LIN {X 0,Y 348.541,Z 887.712,A -85,B 0,C 180,E1 25758,E2 25758} C_VEL
LIN {X 0,Y 309.674,Z 947.389,A -85,B 0,C 180,E1 25764.214,E2 25764.214} C_VEL
LIN {X 0,Y 266.676,Z 997.893,A -85,B 0,C 180,E1 25773.835,E2 25773.835} C_VEL
LIN {X 0,Y 228.973,Z 1035.675,A -85,B 0,C 180,E1 25788.528,E2 25788.528} C_VEL
LIN {X 0,Y 208.44,Z 1057.583,A -85,B 0,C 180,E1 25806.415,E2 25806.415} C_VEL
LIN {X 0,Y 203.021,Z 1066.413,A -85,B 0,C 180,E1 25823.568,E2 25823.568} C_VEL
LIN {X 0,Y 203.129,Z 1067.072,A -85,B 0,C 180,E1 25836.43,E2 25836.43} C_VEL
LIN {X 0,Y 210.406,Z 1057.864,A -85,B 0,C 180,E1 25856.198,E2 25856.198} C_VEL
LIN {X 0,Y 222.858,Z 1046.1,A -85,B 0,C 180,E1 25867.529,E2 25867.529} C_VEL
LIN {X 0,Y 229.777,Z 1035.055,A -85,B 0,C 180,E1 25875.914,E2 25875.914} C_VEL
LIN {X 0,Y 272.123,Z 997.636,A -85,B 0,C 180,E1 25889.741,E2 25889.741} C_VEL
LIN {X 0,Y 318.781,Z 947.378,A -85,B 0,C 180,E1 25898.568,E2 25898.568} C_VEL
LIN {X 0,Y 352.077,Z 901.57,A -85,B 0,C 180,E1 25903.055,E2 25903.055} C_VEL
LIN {X 0,Y 353.093,Z 885.679,A -85,B 0,C 180,E1 25911.32,E2 25911.32} C_VEL
LIN {X 0,Y 353.625,Z 880.392,A -85,B 0,C 180,E1 25918.744,E2 25918.744} C_VEL
LIN {X 0,Y 352.671,Z 887.548,A -85,B 0,C 180,E1 25927.391,E2 25927.391} C_VEL
LIN {X 0,Y 350.818,Z 902.517,A -85,B 0,C 180,E1 25934.441,E2 25934.441} C_VEL
LIN {X 0,Y 306.477,Z 960.307,A -85,B 0,C 180,E1 25940.703,E2 25940.703} C_VEL
LIN {X 0,Y 260.092,Z 1006.735,A -85,B 0,C 180,E1 25950.78,E2 25950.78} C_VEL
LIN {X 0,Y 220.914,Z 1039.817,A -85,B 0,C 180,E1 25966.109,E2 25966.109} C_VEL
LIN {X 0,Y 199.649,Z 1057.963,A -85,B 0,C 180,E1 25985.307,E2 25985.307} C_VEL
LIN {X 0,Y 194.828,Z 1063.462,A -85,B 0,C 180,E1 26003.294,E2 26003.294} C_VEL
LIN {X 0,Y 195.704,Z 1061.786,A -85,B 0,C 180,E1 26016.673,E2 26016.673} C_VEL
LIN {X 0,Y 206.346,Z 1048.693,A -85,B 0,C 180,E1 26037.341,E2 26037.341} C_VEL
LIN {X 0,Y 236.758,Z 1019.964,A -85,B 0,C 180,E1 26055.856,E2 26055.856} C_VEL
LIN {X 0,Y 278.852,Z 977.829,A -85,B 0,C 180,E1 26068.386,E2 26068.386} C_VEL
LIN {X 0,Y 322.725,Z 923.382,A -85,B 0,C 180,E1 26076.469,E2 26076.469} C_VEL
LIN {X 0,Y 342.393,Z 892.633,A -85,B 0,C 180,E1 26079.429,E2 26079.429} C_VEL
LIN {X 0,Y 343.314,Z 872.383,A -85,B 0,C 180,E1 26087.906,E2 26087.906} C_VEL
LIN {X 0,Y 343.606,Z 863.388,A -85,B 0,C 180,E1 26096.228,E2 26096.228} C_VEL
LIN {X 0,Y 343.762,Z 863.668,A -85,B 0,C 180,E1 26101.292,E2 26101.292} C_VEL
LIN {X 0,Y 343.852,Z 876.291,A -85,B 0,C 180,E1 26110.841,E2 26110.841} C_VEL
LIN {X 0,Y 342.839,Z 893.969,A -85,B 0,C 180,E1 26117.448,E2 26117.448} C_VEL
LIN {X 0,Y 301.371,Z 953.407,A -85,B 0,C 180,E1 26123.657,E2 26123.657} C_VEL
LIN {X 0,Y 257.23,Z 1002.52,A -85,B 0,C 180,E1 26133.7,E2 26133.7} C_VEL
LIN {X 0,Y 219.56,Z 1038.628,A -85,B 0,C 180,E1 26148.996,E2 26148.996} C_VEL
LIN {X 0,Y 199.54,Z 1059.052,A -85,B 0,C 180,E1 26167.669,E2 26167.669} C_VEL
LIN {X 0,Y 195.018,Z 1066.321,A -85,B 0,C 180,E1 26183.303,E2 26183.303} C_VEL
LIN {X 0,Y 195.122,Z 1066.998,A -85,B 0,C 180,E1 26196.695,E2 26196.695} C_VEL
LIN {X 0,Y 202.007,Z 1058.771,A -85,B 0,C 180,E1 26215.932,E2 26215.932} C_VEL
LIN {X 0,Y 229.777,Z 1035.055,A -85,B 0,C 180,E1 26235.914,E2 26235.914} C_VEL
LIN {X 0,Y 239.937,Z 1022.061,A -85,B 0,C 180,E1 26243.59,E2 26243.59} C_VEL
LIN {X 0,Y 287.569,Z 978.627,A -85,B 0,C 180,E1 26255.332,E2 26255.332} C_VEL
LIN {X 0,Y 334.687,Z 923.76,A -85,B 0,C 180,E1 26262.455,E2 26262.455} C_VEL
LIN {X 0,Y 347.143,Z 905.9,A -85,B 0,C 180,E1 26263.988,E2 26263.988} C_VEL
LIN {X 0,Y 348.572,Z 891.02,A -85,B 0,C 180,E1 26272.467,E2 26272.467} C_VEL
LIN {X 0,Y 349.117,Z 887.018,A -85,B 0,C 180,E1 26278.727,E2 26278.727} C_VEL
LIN {X 0,Y 347.911,Z 894.709,A -85,B 0,C 180,E1 26287.711,E2 26287.711} C_VEL
LIN {X 0,Y 345.687,Z 907.135,A -85,B 0,C 180,E1 26293.499,E2 26293.499} C_VEL
LIN {X 0,Y 300.619,Z 963.408,A -85,B 0,C 180,E1 26299.715,E2 26299.715} C_VEL
LIN {X 0,Y 253.465,Z 1008.739,A -85,B 0,C 180,E1 26309.829,E2 26309.829} C_VEL
LIN {X 0,Y 212.875,Z 1041.423,A -85,B 0,C 180,E1 26325.724,E2 26325.724} C_VEL
LIN {X 0,Y 191.326,Z 1058.749,A -85,B 0,C 180,E1 26345.704,E2 26345.704} C_VEL
LIN {X 0,Y 186.807,Z 1063.535,A -85,B 0,C 180,E1 26363.005,E2 26363.005} C_VEL
LIN {X 0,Y 187.75,Z 1061.89,A -85,B 0,C 180,E1 26376.957,E2 26376.957} C_VEL
LIN {X 0,Y 197.993,Z 1049.851,A -85,B 0,C 180,E1 26397.274,E2 26397.274} C_VEL
LIN {X 0,Y 227.623,Z 1023.387,A -85,B 0,C 180,E1 26415.862,E2 26415.862} C_VEL
LIN {X 0,Y 270.255,Z 982.815,A -85,B 0,C 180,E1 26428.834,E2 26428.834} C_VEL
LIN {X 0,Y 315.398,Z 929.408,A -85,B 0,C 180,E1 26437.172,E2 26437.172} C_VEL
LIN {X 0,Y 337.365,Z 896.845,A -85,B 0,C 180,E1 26440.31,E2 26440.31} C_VEL
LIN {X 0,Y 338.999,Z 877.413,A -85,B 0,C 180,E1 26449.059,E2 26449.059} C_VEL
LIN {X 0,Y 340.014,Z 868.942,A -85,B 0,C 180,E1 26458.749,E2 26458.749} C_VEL
LIN {X 0,Y 339.391,Z 878.655,A -85,B 0,C 180,E1 26468.385,E2 26468.385} C_VEL
LIN {X 0,Y 338.245,Z 897.158,A -85,B 0,C 180,E1 26476.407,E2 26476.407} C_VEL
LIN {X 0,Y 294.973,Z 956.872,A -85,B 0,C 180,E1 26482.735,E2 26482.735} C_VEL
LIN {X 0,Y 249.571,Z 1005.349,A -85,B 0,C 180,E1 26493.014,E2 26493.014} C_VEL
LIN {X 0,Y 211.634,Z 1040.081,A -85,B 0,C 180,E1 26508.542,E2 26508.542} C_VEL
LIN {X 0,Y 190.684,Z 1060.513,A -85,B 0,C 180,E1 26529.032,E2 26529.032} C_VEL
LIN {X 0,Y 186.999,Z 1067.028,A -85,B 0,C 180,E1 26547.677,E2 26547.677} C_VEL
LIN {X 0,Y 187.65,Z 1065.942,A -85,B 0,C 180,E1 26561.657,E2 26561.657} C_VEL
LIN {X 0,Y 200.399,Z 1053.731,A -85,B 0,C 180,E1 26583.213,E2 26583.213} C_VEL
LIN {X 0,Y 234.442,Z 1026.63,A -85,B 0,C 180,E1 26601.681,E2 26601.681} C_VEL
LIN {X 0,Y 239.937,Z 1022.061,A -85,B 0,C 180,E1 26603.59,E2 26603.59} C_VEL
LIN {X 0,Y 253.584,Z 1007.011,A -85,B 0,C 180,E1 26610.365,E2 26610.365} C_VEL
LIN {X 0,Y 302.812,Z 959.33,A -85,B 0,C 180,E1 26619.879,E2 26619.879} C_VEL
LIN {X 0,Y 342.323,Z 909.562,A -85,B 0,C 180,E1 26625.257,E2 26625.257} C_VEL
LIN {X 0,Y 344.01,Z 896.36,A -85,B 0,C 180,E1 26633.64,E2 26633.64} C_VEL
LIN {X 0,Y 344.292,Z 894.425,A -85,B 0,C 180,E1 26641.236,E2 26641.236} C_VEL
LIN {X 0,Y 342.35,Z 905.549,A -85,B 0,C 180,E1 26650.211,E2 26650.211} C_VEL
LIN {X 0,Y 340.57,Z 911.466,A -85,B 0,C 180,E1 26652.525,E2 26652.525} C_VEL
LIN {X 0,Y 294.571,Z 966.733,A -85,B 0,C 180,E1 26658.74,E2 26658.74} C_VEL
LIN {X 0,Y 245.604,Z 1011.828,A -85,B 0,C 180,E1 26669.183,E2 26669.183} C_VEL
LIN {X 0,Y 204.818,Z 1043.029,A -85,B 0,C 180,E1 26685.302,E2 26685.302} C_VEL
LIN {X 0,Y 182.092,Z 1060.341,A -85,B 0,C 180,E1 26707.99,E2 26707.99} C_VEL
LIN {X 0,Y 179.012,Z 1063.546,A -85,B 0,C 180,E1 26727.983,E2 26727.983} C_VEL
LIN {X 0,Y 182.801,Z 1057.745,A -85,B 0,C 180,E1 26747.458,E2 26747.458} C_VEL
LIN {X 0,Y 204.643,Z 1038.037,A -85,B 0,C 180,E1 26769.038,E2 26769.038} C_VEL
LIN {X 0,Y 244.88,Z 1003.338,A -85,B 0,C 180,E1 26785.134,E2 26785.134} C_VEL
LIN {X 0,Y 291.96,Z 954.998,A -85,B 0,C 180,E1 26795.357,E2 26795.357} C_VEL
LIN {X 0,Y 332.46,Z 900.578,A -85,B 0,C 180,E1 26801.407,E2 26801.407} C_VEL
LIN {X 0,Y 334.388,Z 883.799,A -85,B 0,C 180,E1 26809.302,E2 26809.302} C_VEL
LIN {X 0,Y 335.804,Z 875.772,A -85,B 0,C 180,E1 26818.733,E2 26818.733} C_VEL
LIN {X 0,Y 334.7,Z 885.63,A -85,B 0,C 180,E1 26828.504,E2 26828.504} C_VEL
LIN {X 0,Y 332.665,Z 901.995,A -85,B 0,C 180,E1 26835.463,E2 26835.463} C_VEL
LIN {X 0,Y 288.685,Z 960.322,A -85,B 0,C 180,E1 26841.778,E2 26841.778} C_VEL
LIN {X 0,Y 242.089,Z 1008.031,A -85,B 0,C 180,E1 26852.263,E2 26852.263} C_VEL
LIN {X 0,Y 202.346,Z 1042.515,A -85,B 0,C 180,E1 26868.897,E2 26868.897} C_VEL
LIN {X 0,Y 181.929,Z 1061.643,A -85,B 0,C 180,E1 26890.525,E2 26890.525} C_VEL
LIN {X 0,Y 178.981,Z 1066.945,A -85,B 0,C 180,E1 26907.573,E2 26907.573} C_VEL
LIN {X 0,Y 180.118,Z 1065.434,A -85,B 0,C 180,E1 26924.076,E2 26924.076} C_VEL
LIN {X 0,Y 196.209,Z 1051.677,A -85,B 0,C 180,E1 26946.797,E2 26946.797} C_VEL
LIN {X 0,Y 233.865,Z 1023.081,A -85,B 0,C 180,E1 26964.828,E2 26964.828} C_VEL
LIN {X 0,Y 253.584,Z 1007.011,A -85,B 0,C 180,E1 26970.365,E2 26970.365} C_VEL
LIN {X 0,Y 269.364,Z 989.826,A -85,B 0,C 180,E1 26976.24,E2 26976.24} C_VEL
LIN {X 0,Y 318.309,Z 938.81,A -85,B 0,C 180,E1 26983.774,E2 26983.774} C_VEL
LIN {X 0,Y 337.204,Z 914.36,A -85,B 0,C 180,E1 26986.015,E2 26986.015} C_VEL
LIN {X 0,Y 339.308,Z 901.839,A -85,B 0,C 180,E1 26994.839,E2 26994.839} C_VEL
LIN {X 0,Y 339.456,Z 900.885,A -85,B 0,C 180,E1 27001.253,E2 27001.253} C_VEL
LIN {X 0,Y 337.059,Z 912.229,A -85,B 0,C 180,E1 27010.344,E2 27010.344} C_VEL
LIN {X 0,Y 334.418,Z 917.307,A -85,B 0,C 180,E1 27011.64,E2 27011.64} C_VEL
LIN {X 0,Y 286.994,Z 971.724,A -85,B 0,C 180,E1 27017.993,E2 27017.993} C_VEL
LIN {X 0,Y 237.199,Z 1015.272,A -85,B 0,C 180,E1 27028.634,E2 27028.634} C_VEL
LIN {X 0,Y 195.356,Z 1045.415,A -85,B 0,C 180,E1 27045.683,E2 27045.683} C_VEL
LIN {X 0,Y 174.467,Z 1060.395,A -85,B 0,C 180,E1 27066.974,E2 27066.974} C_VEL
LIN {X 0,Y 170.98,Z 1063.623,A -85,B 0,C 180,E1 27087.959,E2 27087.959} C_VEL
LIN {X 0,Y 174.832,Z 1058.138,A -85,B 0,C 180,E1 27107.671,E2 27107.671} C_VEL
LIN {X 0,Y 197.219,Z 1039.049,A -85,B 0,C 180,E1 27129.877,E2 27129.877} C_VEL
LIN {X 0,Y 239.003,Z 1004.751,A -85,B 0,C 180,E1 27146.381,E2 27146.381} C_VEL
LIN {X 0,Y 287.218,Z 956.934,A -85,B 0,C 180,E1 27156.585,E2 27156.585} C_VEL
LIN {X 0,Y 327.618,Z 904.456,A -85,B 0,C 180,E1 27162.505,E2 27162.505} C_VEL
LIN {X 0,Y 330.043,Z 888.073,A -85,B 0,C 180,E1 27171.051,E2 27171.051} C_VEL
LIN {X 0,Y 331.379,Z 882.482,A -85,B 0,C 180,E1 27178.716,E2 27178.716} C_VEL
LIN {X 0,Y 330.064,Z 891.717,A -85,B 0,C 180,E1 27188.091,E2 27188.091} C_VEL
LIN {X 0,Y 327.626,Z 906.151,A -85,B 0,C 180,E1 27194.438,E2 27194.438} C_VEL
LIN {X 0,Y 281.995,Z 964.279,A -85,B 0,C 180,E1 27200.882,E2 27200.882} C_VEL
LIN {X 0,Y 234.984,Z 1010.175,A -85,B 0,C 180,E1 27211.35,E2 27211.35} C_VEL
LIN {X 0,Y 194.31,Z 1043.843,A -85,B 0,C 180,E1 27228.446,E2 27228.446} C_VEL
LIN {X 0,Y 174.265,Z 1061.532,A -85,B 0,C 180,E1 27249.632,E2 27249.632} C_VEL
LIN {X 0,Y 170.962,Z 1066.863,A -85,B 0,C 180,E1 27267.459,E2 27267.459} C_VEL
LIN {X 0,Y 171.821,Z 1065.811,A -85,B 0,C 180,E1 27282.748,E2 27282.748} C_VEL
LIN {X 0,Y 186.156,Z 1054.082,A -85,B 0,C 180,E1 27305.526,E2 27305.526} C_VEL
LIN {X 0,Y 223.67,Z 1027.273,A -85,B 0,C 180,E1 27324.723,E2 27324.723} C_VEL
LIN {X 0,Y 269.364,Z 989.826,A -85,B 0,C 180,E1 27336.24,E2 27336.24} C_VEL
LIN {X 0,Y 286.604,Z 970.708,A -85,B 0,C 180,E1 27341.286,E2 27341.286} C_VEL
LIN {X 0,Y 332.201,Z 918.868,A -85,B 0,C 180,E1 27346.947,E2 27346.947} C_VEL
LIN {X 0,Y 334.735,Z 907.351,A -85,B 0,C 180,E1 27356.072,E2 27356.072} C_VEL
LIN {X 0,Y 334.247,Z 908.345,A -85,B 0,C 180,E1 27362.574,E2 27362.574} C_VEL
LIN {X 0,Y 331.472,Z 918.963,A -85,B 0,C 180,E1 27370.395,E2 27370.395} C_VEL
LIN {X 0,Y 282.917,Z 973.223,A -85,B 0,C 180,E1 27376.645,E2 27376.645} C_VEL
LIN {X 0,Y 233.296,Z 1015.235,A -85,B 0,C 180,E1 27386.826,E2 27386.826} C_VEL
LIN {X 0,Y 189.349,Z 1045.482,A -85,B 0,C 180,E1 27403.961,E2 27403.961} C_VEL
LIN {X 0,Y 166.924,Z 1060.449,A -85,B 0,C 180,E1 27425.869,E2 27425.869} C_VEL
LIN {X 0,Y 162.944,Z 1063.699,A -85,B 0,C 180,E1 27447.938,E2 27447.938} C_VEL
LIN {X 0,Y 167.135,Z 1058.253,A -85,B 0,C 180,E1 27468.514,E2 27468.514} C_VEL
LIN {X 0,Y 190.412,Z 1039.655,A -85,B 0,C 180,E1 27491.096,E2 27491.096} C_VEL
LIN {X 0,Y 233.243,Z 1006.068,A -85,B 0,C 180,E1 27507.69,E2 27507.69} C_VEL
LIN {X 0,Y 282.722,Z 958.748,A -85,B 0,C 180,E1 27517.871,E2 27517.871} C_VEL
LIN {X 0,Y 322.812,Z 908.34,A -85,B 0,C 180,E1 27523.646,E2 27523.646} C_VEL
LIN {X 0,Y 325.542,Z 893.675,A -85,B 0,C 180,E1 27531.988,E2 27531.988} C_VEL
LIN {X 0,Y 326.852,Z 889.135,A -85,B 0,C 180,E1 27538.698,E2 27538.698} C_VEL
LIN {X 0,Y 325.154,Z 898.537,A -85,B 0,C 180,E1 27548.214,E2 27548.214} C_VEL
LIN {X 0,Y 322.892,Z 909.93,A -85,B 0,C 180,E1 27553.363,E2 27553.363} C_VEL
LIN {X 0,Y 276.004,Z 967.263,A -85,B 0,C 180,E1 27559.803,E2 27559.803} C_VEL
LIN {X 0,Y 226.78,Z 1013.301,A -85,B 0,C 180,E1 27570.722,E2 27570.722} C_VEL
LIN {X 0,Y 186.449,Z 1045.048,A -85,B 0,C 180,E1 27587.859,E2 27587.859} C_VEL
LIN {X 0,Y 165.492,Z 1062.651,A -85,B 0,C 180,E1 27611.296,E2 27611.296} C_VEL
LIN {X 0,Y 163.159,Z 1067.062,A -85,B 0,C 180,E1 27632.665,E2 27632.665} C_VEL
LIN {X 0,Y 167.989,Z 1062.223,A -85,B 0,C 180,E1 27653.968,E2 27653.968} C_VEL
LIN {X 0,Y 196.071,Z 1043.127,A -85,B 0,C 180,E1 27677.286,E2 27677.286} C_VEL
LIN {X 0,Y 242.567,Z 1009.611,A -85,B 0,C 180,E1 27692.981,E2 27692.981} C_VEL
LIN {X 0,Y 286.604,Z 970.708,A -85,B 0,C 180,E1 27701.286,E2 27701.286} C_VEL
LIN {X 0,Y 304.813,Z 949.598,A -85,B 0,C 180,E1 27705.556,E2 27705.556} C_VEL
LIN {X 0,Y 327.39,Z 922.805,A -85,B 0,C 180,E1 27708.249,E2 27708.249} C_VEL
LIN {X 0,Y 329.635,Z 913.664,A -85,B 0,C 180,E1 27716.011,E2 27716.011} C_VEL
LIN {X 0,Y 329.018,Z 914.821,A -85,B 0,C 180,E1 27722.845,E2 27722.845} C_VEL
LIN {X 0,Y 326.672,Z 923.17,A -85,B 0,C 180,E1 27729.33,E2 27729.33} C_VEL
LIN {X 0,Y 275.725,Z 977.559,A -85,B 0,C 180,E1 27735.748,E2 27735.748} C_VEL
LIN {X 0,Y 223.661,Z 1019.345,A -85,B 0,C 180,E1 27746.502,E2 27746.502} C_VEL
LIN {X 0,Y 179.921,Z 1047.733,A -85,B 0,C 180,E1 27764.241,E2 27764.241} C_VEL
LIN {X 0,Y 159.422,Z 1060.503,A -85,B 0,C 180,E1 27784.655,E2 27784.655} C_VEL
LIN {X 0,Y 154.915,Z 1063.776,A -85,B 0,C 180,E1 27807.919,E2 27807.919} C_VEL
LIN {X 0,Y 159.467,Z 1058.368,A -85,B 0,C 180,E1 27829.439,E2 27829.439} C_VEL
LIN {X 0,Y 186.264,Z 1038.517,A -85,B 0,C 180,E1 27853.787,E2 27853.787} C_VEL
LIN {X 0,Y 231.752,Z 1004.007,A -85,B 0,C 180,E1 27870.108,E2 27870.108} C_VEL
LIN {X 0,Y 282.667,Z 955.853,A -85,B 0,C 180,E1 27879.852,E2 27879.852} C_VEL
LIN {X 0,Y 317.979,Z 912.169,A -85,B 0,C 180,E1 27884.811,E2 27884.811} C_VEL
LIN {X 0,Y 320.895,Z 898.962,A -85,B 0,C 180,E1 27893.239,E2 27893.239} C_VEL
LIN {X 0,Y 322.215,Z 895.711,A -85,B 0,C 180,E1 27898.68,E2 27898.68} C_VEL
LIN {X 0,Y 320.143,Z 905.118,A -85,B 0,C 180,E1 27908.207,E2 27908.207} C_VEL
LIN {X 0,Y 318.121,Z 913.642,A -85,B 0,C 180,E1 27912.264,E2 27912.264} C_VEL
LIN {X 0,Y 269.714,Z 970.668,A -85,B 0,C 180,E1 27918.751,E2 27918.751} C_VEL
LIN {X 0,Y 220.53,Z 1014.822,A -85,B 0,C 180,E1 27929.474,E2 27929.474} C_VEL
LIN {X 0,Y 178.285,Z 1046.464,A -85,B 0,C 180,E1 27947.407,E2 27947.407} C_VEL
LIN {X 0,Y 157.783,Z 1062.539,A -85,B 0,C 180,E1 27970.345,E2 27970.345} C_VEL
LIN {X 0,Y 155.149,Z 1066.988,A -85,B 0,C 180,E1 27992.802,E2 27992.802} C_VEL
LIN {X 0,Y 161.499,Z 1061.503,A -85,B 0,C 180,E1 28016.64,E2 28016.64} C_VEL
LIN {X 0,Y 193.898,Z 1041.055,A -85,B 0,C 180,E1 28040.633,E2 28040.633} C_VEL
LIN {X 0,Y 241.83,Z 1007.483,A -85,B 0,C 180,E1 28055.402,E2 28055.402} C_VEL
LIN {X 0,Y 293.56,Z 961.468,A -85,B 0,C 180,E1 28064.14,E2 28064.14} C_VEL
LIN {X 0,Y 304.813,Z 949.598,A -85,B 0,C 180,E1 28065.556,E2 28065.556} C_VEL
LIN {X 0,Y 315.848,Z 935.192,A -85,B 0,C 180,E1 28068.457,E2 28068.457} C_VEL
LIN {X 0,Y 322.477,Z 926.683,A -85,B 0,C 180,E1 28069.633,E2 28069.633} C_VEL
LIN {X 0,Y 324.901,Z 918.901,A -85,B 0,C 180,E1 28078.633,E2 28078.633} C_VEL
LIN {X 0,Y 322.004,Z 926.631,A -85,B 0,C 180,E1 28087.756,E2 28087.756} C_VEL
LIN {X 0,Y 308.073,Z 943.178,A -85,B 0,C 180,E1 28089.688,E2 28089.688} C_VEL
LIN {X 0,Y 255.938,Z 992.544,A -85,B 0,C 180,E1 28096.864,E2 28096.864} C_VEL
LIN {X 0,Y 203.521,Z 1030.156,A -85,B 0,C 180,E1 28109.295,E2 28109.295} C_VEL
LIN {X 0,Y 163.638,Z 1053.752,A -85,B 0,C 180,E1 28129.556,E2 28129.556} C_VEL
LIN {X 0,Y 147.501,Z 1063.35,A -85,B 0,C 180,E1 28155.105,E2 28155.105} C_VEL
LIN {X 0,Y 147.384,Z 1063.425,A -85,B 0,C 180,E1 28172.947,E2 28172.947} C_VEL
LIN {X 0,Y 157.662,Z 1054.167,A -85,B 0,C 180,E1 28198.743,E2 28198.743} C_VEL
LIN {X 0,Y 193.927,Z 1029.509,A -85,B 0,C 180,E1 28221.542,E2 28221.542} C_VEL
LIN {X 0,Y 243.759,Z 990.885,A -85,B 0,C 180,E1 28235.33,E2 28235.33} C_VEL
LIN {X 0,Y 294.684,Z 939.802,A -85,B 0,C 180,E1 28243.364,E2 28243.364} C_VEL
LIN {X 0,Y 312.988,Z 916.85,A -85,B 0,C 180,E1 28245.651,E2 28245.651} C_VEL
LIN {X 0,Y 315.997,Z 905.548,A -85,B 0,C 180,E1 28253.133,E2 28253.133} C_VEL
LIN {X 0,Y 317.387,Z 902.16,A -85,B 0,C 180,E1 28258.66,E2 28258.66} C_VEL
LIN {X 0,Y 314.948,Z 911.829,A -85,B 0,C 180,E1 28268.344,E2 28268.344} C_VEL
LIN {X 0,Y 312.896,Z 918.131,A -85,B 0,C 180,E1 28271.196,E2 28271.196} C_VEL
LIN {X 0,Y 264.084,Z 973.512,A -85,B 0,C 180,E1 28277.564,E2 28277.564} C_VEL
LIN {X 0,Y 213.382,Z 1017.086,A -85,B 0,C 180,E1 28288.427,E2 28288.427} C_VEL
LIN {X 0,Y 172.011,Z 1046.481,A -85,B 0,C 180,E1 28305.696,E2 28305.696} C_VEL
LIN {X 0,Y 150.114,Z 1062.427,A -85,B 0,C 180,E1 28329.296,E2 28329.296} C_VEL
LIN {X 0,Y 147.122,Z 1066.915,A -85,B 0,C 180,E1 28352.955,E2 28352.955} C_VEL
LIN {X 0,Y 154.196,Z 1061.456,A -85,B 0,C 180,E1 28378.01,E2 28378.01} C_VEL
LIN {X 0,Y 187.676,Z 1041.663,A -85,B 0,C 180,E1 28402.135,E2 28402.135} C_VEL
LIN {X 0,Y 238.513,Z 1007.525,A -85,B 0,C 180,E1 28417.204,E2 28417.204} C_VEL
LIN {X 0,Y 292.633,Z 960.34,A -85,B 0,C 180,E1 28425.833,E2 28425.833} C_VEL
LIN {X 0,Y 315.848,Z 935.192,A -85,B 0,C 180,E1 28428.457,E2 28428.457} C_VEL
LIN {X 0,Y 318.528,Z 930.466,A -85,B 0,C 180,E1 28430.192,E2 28430.192} C_VEL
LIN {X 0,Y 318.15,Z 928.9,A -85,B 0,C 180,E1 28432.623,E2 28432.623} C_VEL
LIN {X 0,Y 319.703,Z 924.997,A -85,B 0,C 180,E1 28438.61,E2 28438.61} C_VEL
LIN {X 0,Y 316.908,Z 931.413,A -85,B 0,C 180,E1 28446.847,E2 28446.847} C_VEL
LIN {X 0,Y 264.503,Z 983.599,A -85,B 0,C 180,E1 28453.366,E2 28453.366} C_VEL
LIN {X 0,Y 208.506,Z 1024.582,A -85,B 0,C 180,E1 28464.617,E2 28464.617} C_VEL
LIN {X 0,Y 164.61,Z 1049.936,A -85,B 0,C 180,E1 28482.528,E2 28482.528} C_VEL
LIN {X 0,Y 141.564,Z 1062.315,A -85,B 0,C 180,E1 28507.979,E2 28507.979} C_VEL
LIN {X 0,Y 139.41,Z 1063.518,A -85,B 0,C 180,E1 28533.116,E2 28533.116} C_VEL
LIN {X 0,Y 150.434,Z 1054.39,A -85,B 0,C 180,E1 28560.053,E2 28560.053} C_VEL
LIN {X 0,Y 187.275,Z 1030.854,A -85,B 0,C 180,E1 28582.847,E2 28582.847} C_VEL
LIN {X 0,Y 237.613,Z 993.563,A -85,B 0,C 180,E1 28596.545,E2 28596.545} C_VEL
LIN {X 0,Y 289.173,Z 943.824,A -85,B 0,C 180,E1 28604.486,E2 28604.486} C_VEL
LIN {X 0,Y 308.283,Z 920.824,A -85,B 0,C 180,E1 28606.87,E2 28606.87} C_VEL
LIN {X 0,Y 311.278,Z 910.703,A -85,B 0,C 180,E1 28614.813,E2 28614.813} C_VEL
LIN {X 0,Y 312.545,Z 908.591,A -85,B 0,C 180,E1 28618.639,E2 28618.639} C_VEL
LIN {X 0,Y 309.803,Z 917.558,A -85,B 0,C 180,E1 28627.969,E2 28627.969} C_VEL
LIN {X 0,Y 307.534,Z 922.918,A -85,B 0,C 180,E1 28630.094,E2 28630.094} C_VEL
LIN {X 0,Y 258.176,Z 976.584,A -85,B 0,C 180,E1 28636.371,E2 28636.371} C_VEL
LIN {X 0,Y 205.301,Z 1019.863,A -85,B 0,C 180,E1 28647.583,E2 28647.583} C_VEL
LIN {X 0,Y 161.097,Z 1049.48,A -85,B 0,C 180,E1 28666.967,E2 28666.967} C_VEL
LIN {X 0,Y 140.277,Z 1064.273,A -85,B 0,C 180,E1 28694.322,E2 28694.322} C_VEL
LIN {X 0,Y 139.123,Z 1066.841,A -85,B 0,C 180,E1 28713.126,E2 28713.126} C_VEL
LIN {X 0,Y 148.009,Z 1060.859,A -85,B 0,C 180,E1 28740.817,E2 28740.817} C_VEL
LIN {X 0,Y 185.346,Z 1040.207,A -85,B 0,C 180,E1 28765.236,E2 28765.236} C_VEL
LIN {X 0,Y 238.487,Z 1005.268,A -85,B 0,C 180,E1 28779.644,E2 28779.644} C_VEL
LIN {X 0,Y 292.944,Z 958.208,A -85,B 0,C 180,E1 28787.657,E2 28787.657} C_VEL
LIN {X 0,Y 317.219,Z 931.772,A -85,B 0,C 180,E1 28790.33,E2 28790.33} C_VEL
LIN {X 0,Y 318.15,Z 928.9,A -85,B 0,C 180,E1 28792.623,E2 28792.623} C_VEL
LIN {X 0,Y 314.16,Z 931.145,A -85,B 0,C 180,E1 28799.042,E2 28799.042} C_VEL
LIN {X 0,Y 310.88,Z 937.358,A -85,B 0,C 180,E1 28806.139,E2 28806.139} C_VEL
LIN {X 0,Y 256.296,Z 988.669,A -85,B 0,C 180,E1 28812.509,E2 28812.509} C_VEL
LIN {X 0,Y 199.532,Z 1027.899,A -85,B 0,C 180,E1 28823.989,E2 28823.989} C_VEL
LIN {X 0,Y 153.017,Z 1052.894,A -85,B 0,C 180,E1 28844.18,E2 28844.18} C_VEL
LIN {X 0,Y 133.976,Z 1062.369,A -85,B 0,C 180,E1 28866.661,E2 28866.661} C_VEL
LIN {X 0,Y 130.82,Z 1064.003,A -85,B 0,C 180,E1 28887.897,E2 28887.897} C_VEL
LIN {X 0,Y 136.819,Z 1058.712,A -85,B 0,C 180,E1 28912.823,E2 28912.823} C_VEL
LIN {X 0,Y 169.445,Z 1038.993,A -85,B 0,C 180,E1 28939.523,E2 28939.523} C_VEL
LIN {X 0,Y 218.959,Z 1005.893,A -85,B 0,C 180,E1 28955.288,E2 28955.288} C_VEL
LIN {X 0,Y 273.528,Z 958.465,A -85,B 0,C 180,E1 28964.394,E2 28964.394} C_VEL
LIN {X 0,Y 302.6,Z 926.182,A -85,B 0,C 180,E1 28967.738,E2 28967.738} C_VEL
LIN {X 0,Y 306.017,Z 917.282,A -85,B 0,C 180,E1 28974.338,E2 28974.338} C_VEL
LIN {X 0,Y 307.424,Z 914.825,A -85,B 0,C 180,E1 28978.616,E2 28978.616} C_VEL
LIN {X 0,Y 304.325,Z 924.217,A -85,B 0,C 180,E1 28988.144,E2 28988.144} C_VEL
LIN {X 0,Y 300.883,Z 929.007,A -85,B 0,C 180,E1 28989.101,E2 28989.101} C_VEL
LIN {X 0,Y 249.821,Z 981.791,A -85,B 0,C 180,E1 28995.514,E2 28995.514} C_VEL
LIN {X 0,Y 195.876,Z 1023.63,A -85,B 0,C 180,E1 29007.092,E2 29007.092} C_VEL
LIN {X 0,Y 151.428,Z 1051.648,A -85,B 0,C 180,E1 29027.474,E2 29027.474} C_VEL
LIN {X 0,Y 132.478,Z 1064.171,A -85,B 0,C 180,E1 29053.373,E2 29053.373} C_VEL
LIN {X 0,Y 131.093,Z 1066.767,A -85,B 0,C 180,E1 29073.317,E2 29073.317} C_VEL
LIN {X 0,Y 141.018,Z 1060.812,A -85,B 0,C 180,E1 29102.527,E2 29102.527} C_VEL
LIN {X 0,Y 181.078,Z 1040.013,A -85,B 0,C 180,E1 29127.544,E2 29127.544} C_VEL
LIN {X 0,Y 235.796,Z 1005.271,A -85,B 0,C 180,E1 29141.549,E2 29141.549} C_VEL
LIN {X 0,Y 291.677,Z 957.947,A -85,B 0,C 180,E1 29149.276,E2 29149.276} C_VEL
LIN {X 0,Y 312.177,Z 936.371,A -85,B 0,C 180,E1 29151.425,E2 29151.425} C_VEL
LIN {X 0,Y 314.16,Z 931.145,A -85,B 0,C 180,E1 29159.042,E2 29159.042} C_VEL
LIN {X 0,Y 307.409,Z 939.206,A -85,B 0,C 180,E1 29163.019,E2 29163.019} C_VEL
LIN {X 0,Y 304.604,Z 943.034,A -85,B 0,C 180,E1 29165.11,E2 29165.11} C_VEL
LIN {X 0,Y 249.444,Z 992.595,A -85,B 0,C 180,E1 29171.397,E2 29171.397} C_VEL
LIN {X 0,Y 193.005,Z 1029.769,A -85,B 0,C 180,E1 29182.602,E2 29182.602} C_VEL
LIN {X 0,Y 144.262,Z 1054.348,A -85,B 0,C 180,E1 29203.985,E2 29203.985} C_VEL
LIN {X 0,Y 123.998,Z 1063.542,A -85,B 0,C 180,E1 29232.196,E2 29232.196} C_VEL
LIN {X 0,Y 123.4,Z 1063.705,A -85,B 0,C 180,E1 29253.521,E2 29253.521} C_VEL
LIN {X 0,Y 137.279,Z 1054.308,A -85,B 0,C 180,E1 29284.104,E2 29284.104} C_VEL
LIN {X 0,Y 179.486,Z 1030.158,A -85,B 0,C 180,E1 29307.655,E2 29307.655} C_VEL
LIN {X 0,Y 233.202,Z 992.722,A -85,B 0,C 180,E1 29320.537,E2 29320.537} C_VEL
LIN {X 0,Y 286.991,Z 942.531,A -85,B 0,C 180,E1 29327.822,E2 29327.822} C_VEL
LIN {X 0,Y 298.604,Z 929.027,A -85,B 0,C 180,E1 29329.348,E2 29329.348} C_VEL
LIN {X 0,Y 302.291,Z 921.071,A -85,B 0,C 180,E1 29338.593,E2 29338.593} C_VEL
LIN {X 0,Y 299.148,Z 929.067,A -85,B 0,C 180,E1 29347.319,E2 29347.319} C_VEL
LIN {X 0,Y 246.046,Z 983.018,A -85,B 0,C 180,E1 29353.91,E2 29353.91} C_VEL
LIN {X 0,Y 190.338,Z 1024.723,A -85,B 0,C 180,E1 29365.413,E2 29365.413} C_VEL
LIN {X 0,Y 143.539,Z 1052.496,A -85,B 0,C 180,E1 29386.633,E2 29386.633} C_VEL
LIN {X 0,Y 124.701,Z 1064.069,A -85,B 0,C 180,E1 29412.303,E2 29412.303} C_VEL
LIN {X 0,Y 123.078,Z 1066.692,A -85,B 0,C 180,E1 29433.534,E2 29433.534} C_VEL
LIN {X 0,Y 134.139,Z 1060.765,A -85,B 0,C 180,E1 29464.421,E2 29464.421} C_VEL
LIN {X 0,Y 175.927,Z 1040.414,A -85,B 0,C 180,E1 29489.539,E2 29489.539} C_VEL
LIN {X 0,Y 233.31,Z 1005.325,A -85,B 0,C 180,E1 29503.476,E2 29503.476} C_VEL
LIN {X 0,Y 289.915,Z 958.411,A -85,B 0,C 180,E1 29510.829,E2 29510.829} C_VEL
LIN {X 0,Y 307.108,Z 940.558,A -85,B 0,C 180,E1 29512.872,E2 29512.872} C_VEL
LIN {X 0,Y 308.779,Z 937.059,A -85,B 0,C 180,E1 29518.903,E2 29518.903} C_VEL
LIN {X 0,Y 307.409,Z 939.206,A -85,B 0,C 180,E1 29523.019,E2 29523.019} C_VEL
LIN {X 0,Y 301.336,Z 945.844,A -85,B 0,C 180,E1 29524.181,E2 29524.181} C_VEL
LIN {X 0,Y 291.695,Z 955.246,A -85,B 0,C 180,E1 29524.641,E2 29524.641} C_VEL
LIN {X 0,Y 233.567,Z 1002.85,A -85,B 0,C 180,E1 29531.565,E2 29531.565} C_VEL
LIN {X 0,Y 174.923,Z 1037.606,A -85,B 0,C 180,E1 29544.457,E2 29544.457} C_VEL
LIN {X 0,Y 132.185,Z 1057.015,A -85,B 0,C 180,E1 29566.501,E2 29566.501} C_VEL
LIN {X 0,Y 114.855,Z 1064.198,A -85,B 0,C 180,E1 29598.576,E2 29598.576} C_VEL
LIN {X 0,Y 116.276,Z 1062.783,A -85,B 0,C 180,E1 29621.279,E2 29621.279} C_VEL
LIN {X 0,Y 136.972,Z 1051.023,A -85,B 0,C 180,E1 29651.623,E2 29651.623} C_VEL
LIN {X 0,Y 184.296,Z 1024.854,A -85,B 0,C 180,E1 29672.702,E2 29672.702} C_VEL
LIN {X 0,Y 241.357,Z 984.418,A -85,B 0,C 180,E1 29684.097,E2 29684.097} C_VEL
LIN {X 0,Y 292.926,Z 934.616,A -85,B 0,C 180,E1 29690.143,E2 29690.143} C_VEL
LIN {X 0,Y 296.954,Z 927.131,A -85,B 0,C 180,E1 29698.567,E2 29698.567} C_VEL
LIN {X 0,Y 293.433,Z 934.571,A -85,B 0,C 180,E1 29706.456,E2 29706.456} C_VEL
LIN {X 0,Y 240.76,Z 985.732,A -85,B 0,C 180,E1 29712.513,E2 29712.513} C_VEL
LIN {X 0,Y 183.669,Z 1026.471,A -85,B 0,C 180,E1 29723.969,E2 29723.969} C_VEL
LIN {X 0,Y 134.845,Z 1053.783,A -85,B 0,C 180,E1 29746.357,E2 29746.357} C_VEL
LIN {X 0,Y 116.979,Z 1063.966,A -85,B 0,C 180,E1 29771.092,E2 29771.092} C_VEL
LIN {X 0,Y 115.048,Z 1066.616,A -85,B 0,C 180,E1 29793.781,E2 29793.781} C_VEL
LIN {X 0,Y 127.436,Z 1060.719,A -85,B 0,C 180,E1 29826.513,E2 29826.513} C_VEL
LIN {X 0,Y 171.855,Z 1040.409,A -85,B 0,C 180,E1 29851.933,E2 29851.933} C_VEL
LIN {X 0,Y 231.098,Z 1005.379,A -85,B 0,C 180,E1 29865.438,E2 29865.438} C_VEL
LIN {X 0,Y 289.689,Z 957.591,A -85,B 0,C 180,E1 29872.528,E2 29872.528} C_VEL
LIN {X 0,Y 301.837,Z 945.318,A -85,B 0,C 180,E1 29873.923,E2 29873.923} C_VEL
LIN {X 0,Y 303.253,Z 942.672,A -85,B 0,C 180,E1 29878.535,E2 29878.535} C_VEL
LIN {X 0,Y 300.237,Z 946.813,A -85,B 0,C 180,E1 29883.881,E2 29883.881} C_VEL
LIN {X 0,Y 291.695,Z 955.246,A -85,B 0,C 180,E1 29884.641,E2 29884.641} C_VEL
LIN {X 0,Y 264.974,Z 978.254,A -85,B 0,C 180,E1 29885.484,E2 29885.484} C_VEL
LIN {X 0,Y 203.479,Z 1020.693,A -85,B 0,C 180,E1 29894.35,E2 29894.35} C_VEL
LIN {X 0,Y 146.527,Z 1048.983,A -85,B 0,C 180,E1 29911.449,E2 29911.449} C_VEL
LIN {X 0,Y 111.559,Z 1062.609,A -85,B 0,C 180,E1 29941.99,E2 29941.99} C_VEL
LIN {X 0,Y 107.417,Z 1063.891,A -85,B 0,C 180,E1 29974.046,E2 29974.046} C_VEL
LIN {X 0,Y 123.898,Z 1054.651,A -85,B 0,C 180,E1 30008.141,E2 30008.141} C_VEL
LIN {X 0,Y 171.245,Z 1030.524,A -85,B 0,C 180,E1 30032.313,E2 30032.313} C_VEL
LIN {X 0,Y 228.281,Z 993.192,A -85,B 0,C 180,E1 30044.404,E2 30044.404} C_VEL
LIN {X 0,Y 284.013,Z 943.128,A -85,B 0,C 180,E1 30051.022,E2 30051.022} C_VEL
LIN {X 0,Y 288.744,Z 937.901,A -85,B 0,C 180,E1 30051.826,E2 30051.826} C_VEL
LIN {X 0,Y 291.548,Z 933.134,A -85,B 0,C 180,E1 30058.541,E2 30058.541} C_VEL
LIN {X 0,Y 288.148,Z 939.219,A -85,B 0,C 180,E1 30065.247,E2 30065.247} C_VEL
LIN {X 0,Y 232.495,Z 990.657,A -85,B 0,C 180,E1 30071.481,E2 30071.481} C_VEL
LIN {X 0,Y 173.521,Z 1030.296,A -85,B 0,C 180,E1 30083.425,E2 30083.425} C_VEL
LIN {X 0,Y 126.715,Z 1054.785,A -85,B 0,C 180,E1 30105.591,E2 30105.591} C_VEL
LIN {X 0,Y 107.397,Z 1065.308,A -85,B 0,C 180,E1 30137.774,E2 30137.774} C_VEL
LIN {X 0,Y 107.474,Z 1066.184,A -85,B 0,C 180,E1 30162.221,E2 30162.221} C_VEL
LIN {X 0,Y 127.129,Z 1058.164,A -85,B 0,C 180,E1 30194.603,E2 30194.603} C_VEL
LIN {X 0,Y 178.082,Z 1035.368,A -85,B 0,C 180,E1 30217.39,E2 30217.39} C_VEL
LIN {X 0,Y 239.54,Z 998.238,A -85,B 0,C 180,E1 30228.886,E2 30228.886} C_VEL
LIN {X 0,Y 296.588,Z 950.125,A -85,B 0,C 180,E1 30235.042,E2 30235.042} C_VEL
LIN {X 0,Y 296.757,Z 949.505,A -85,B 0,C 180,E1 30241.434,E2 30241.434} C_VEL
LIN {X 0,Y 294.386,Z 952.034,A -85,B 0,C 180,E1 30242.732,E2 30242.732} C_VEL
LIN {X 0,Y 264.974,Z 978.254,A -85,B 0,C 180,E1 30245.484,E2 30245.484} C_VEL
LIN {X 0,Y 236.573,Z 998.829,A -85,B 0,C 180,E1 30246.739,E2 30246.739} C_VEL
LIN {X 0,Y 174.971,Z 1034.525,A -85,B 0,C 180,E1 30257.618,E2 30257.618} C_VEL
LIN {X 0,Y 120.616,Z 1057.084,A -85,B 0,C 180,E1 30281.03,E2 30281.03} C_VEL
LIN {X 0,Y 98.981,Z 1064.345,A -85,B 0,C 180,E1 30316.712,E2 30316.712} C_VEL
LIN {X 0,Y 100.571,Z 1062.969,A -85,B 0,C 180,E1 30343.07,E2 30343.07} C_VEL
LIN {X 0,Y 125.219,Z 1051.295,A -85,B 0,C 180,E1 30376.6,E2 30376.6} C_VEL
LIN {X 0,Y 178.747,Z 1024.464,A -85,B 0,C 180,E1 30397.748,E2 30397.748} C_VEL
LIN {X 0,Y 238.341,Z 984.137,A -85,B 0,C 180,E1 30408.012,E2 30408.012} C_VEL
LIN {X 0,Y 282.866,Z 943.425,A -85,B 0,C 180,E1 30412.636,E2 30412.636} C_VEL
LIN {X 0,Y 286.007,Z 939.037,A -85,B 0,C 180,E1 30418.512,E2 30418.512} C_VEL
LIN {X 0,Y 283.319,Z 943.324,A -85,B 0,C 180,E1 30423.952,E2 30423.952} C_VEL
LIN {X 0,Y 227.066,Z 993.42,A -85,B 0,C 180,E1 30429.993,E2 30429.993} C_VEL
LIN {X 0,Y 167.287,Z 1031.881,A -85,B 0,C 180,E1 30441.703,E2 30441.703} C_VEL
LIN {X 0,Y 118.154,Z 1055.984,A -85,B 0,C 180,E1 30465.102,E2 30465.102} C_VEL
LIN {X 0,Y 99.512,Z 1065.215,A -85,B 0,C 180,E1 30496.789,E2 30496.789} C_VEL
LIN {X 0,Y 99.578,Z 1066.11,A -85,B 0,C 180,E1 30523.206,E2 30523.206} C_VEL
LIN {X 0,Y 121.9,Z 1057.928,A -85,B 0,C 180,E1 30557.748,E2 30557.748} C_VEL
LIN {X 0,Y 177.117,Z 1034.361,A -85,B 0,C 180,E1 30580.438,E2 30580.438} C_VEL
LIN {X 0,Y 239.857,Z 997.096,A -85,B 0,C 180,E1 30591.06,E2 30591.06} C_VEL
LIN {X 0,Y 291.045,Z 954.917,A -85,B 0,C 180,E1 30596.201,E2 30596.201} C_VEL
LIN {X 0,Y 291.222,Z 954.441,A -85,B 0,C 180,E1 30599.968,E2 30599.968} C_VEL
LIN {X 0,Y 288.269,Z 957.399,A -85,B 0,C 180,E1 30601.578,E2 30601.578} C_VEL
LIN {X 0,Y 236.573,Z 998.829,A -85,B 0,C 180,E1 30606.739,E2 30606.739} C_VEL
LIN {X 0,Y 206.764,Z 1016.838,A -85,B 0,C 180,E1 30608.561,E2 30608.561} C_VEL
LIN {X 0,Y 144.131,Z 1046.75,A -85,B 0,C 180,E1 30623.212,E2 30623.212} C_VEL
LIN {X 0,Y 103.432,Z 1060.931,A -85,B 0,C 180,E1 30648.717,E2 30648.717} C_VEL
LIN {X 0,Y 90.649,Z 1064.509,A -85,B 0,C 180,E1 30685.2,E2 30685.2} C_VEL
LIN {X 0,Y 98.069,Z 1060.474,A -85,B 0,C 180,E1 30717.636,E2 30717.636} C_VEL
LIN {X 0,Y 140.526,Z 1042.425,A -85,B 0,C 180,E1 30749.684,E2 30749.684} C_VEL
LIN {X 0,Y 201.79,Z 1009.115,A -85,B 0,C 180,E1 30765.138,E2 30765.138} C_VEL
LIN {X 0,Y 261.907,Z 963.206,A -85,B 0,C 180,E1 30772.527,E2 30772.527} C_VEL
LIN {X 0,Y 278.428,Z 947.303,A -85,B 0,C 180,E1 30774.196,E2 30774.196} C_VEL
LIN {X 0,Y 280.327,Z 944.794,A -85,B 0,C 180,E1 30778.482,E2 30778.482} C_VEL
LIN {X 0,Y 277.746,Z 948.362,A -85,B 0,C 180,E1 30782.685,E2 30782.685} C_VEL
LIN {X 0,Y 220.459,Z 997.147,A -85,B 0,C 180,E1 30788.599,E2 30788.599} C_VEL
LIN {X 0,Y 159.948,Z 1033.963,A -85,B 0,C 180,E1 30800.18,E2 30800.18} C_VEL
LIN {X 0,Y 108.199,Z 1057.541,A -85,B 0,C 180,E1 30825.817,E2 30825.817} C_VEL
LIN {X 0,Y 91.638,Z 1065.122,A -85,B 0,C 180,E1 30855.63,E2 30855.63} C_VEL
LIN {X 0,Y 91.702,Z 1066.036,A -85,B 0,C 180,E1 30884.364,E2 30884.364} C_VEL
LIN {X 0,Y 116.939,Z 1057.733,A -85,B 0,C 180,E1 30921.086,E2 30921.086} C_VEL
LIN {X 0,Y 173.779,Z 1034.709,A -85,B 0,C 180,E1 30942.849,E2 30942.849} C_VEL
LIN {X 0,Y 238.709,Z 997.153,A -85,B 0,C 180,E1 30953.026,E2 30953.026} C_VEL
LIN {X 0,Y 285.469,Z 959.853,A -85,B 0,C 180,E1 30957.392,E2 30957.392} C_VEL
LIN {X 0,Y 284.352,Z 960.825,A -85,B 0,C 180,E1 30960.223,E2 30960.223} C_VEL
LIN {X 0,Y 224.312,Z 1006.324,A -85,B 0,C 180,E1 30966.093,E2 30966.093} C_VEL
LIN {X 0,Y 206.764,Z 1016.838,A -85,B 0,C 180,E1 30968.561,E2 30968.561} C_VEL
LIN {X 0,Y 175.876,Z 1032.156,A -85,B 0,C 180,E1 30971.18,E2 30971.18} C_VEL
LIN {X 0,Y 115.396,Z 1055.594,A -85,B 0,C 180,E1 30991.33,E2 30991.33} C_VEL
LIN {X 0,Y 85.943,Z 1063.863,A -85,B 0,C 180,E1 31023.823,E2 31023.823} C_VEL
LIN {X 0,Y 83.447,Z 1064.169,A -85,B 0,C 180,E1 31055.211,E2 31055.211} C_VEL
LIN {X 0,Y 105.327,Z 1055.169,A -85,B 0,C 180,E1 31096.04,E2 31096.04} C_VEL
LIN {X 0,Y 161.285,Z 1031.07,A -85,B 0,C 180,E1 31120.082,E2 31120.082} C_VEL
LIN {X 0,Y 224.731,Z 992.577,A -85,B 0,C 180,E1 31130.691,E2 31130.691} C_VEL
LIN {X 0,Y 272.368,Z 952.84,A -85,B 0,C 180,E1 31135.24,E2 31135.24} C_VEL
LIN {X 0,Y 273.978,Z 951.261,A -85,B 0,C 180,E1 31140.034,E2 31140.034} C_VEL
LIN {X 0,Y 272.453,Z 952.956,A -85,B 0,C 180,E1 31141.351,E2 31141.351} C_VEL
LIN {X 0,Y 212.136,Z 1001.806,A -85,B 0,C 180,E1 31147.338,E2 31147.338} C_VEL
LIN {X 0,Y 148.89,Z 1037.851,A -85,B 0,C 180,E1 31159.602,E2 31159.602} C_VEL
LIN {X 0,Y 98.617,Z 1058.925,A -85,B 0,C 180,E1 31186.218,E2 31186.218} C_VEL
LIN {X 0,Y 82.806,Z 1065.953,A -85,B 0,C 180,E1 31224.749,E2 31224.749} C_VEL
LIN {X 0,Y 86.835,Z 1065.094,A -85,B 0,C 180,E1 31255.888,E2 31255.888} C_VEL
LIN {X 0,Y 128.035,Z 1052.363,A -85,B 0,C 180,E1 31292.661,E2 31292.661} C_VEL
LIN {X 0,Y 192.896,Z 1024.253,A -85,B 0,C 180,E1 31309.32,E2 31309.32} C_VEL
LIN {X 0,Y 258.648,Z 982.062,A -85,B 0,C 180,E1 31316.901,E2 31316.901} C_VEL
LIN {X 0,Y 279.698,Z 964.842,A -85,B 0,C 180,E1 31318.812,E2 31318.812} C_VEL
LIN {X 0,Y 216.845,Z 1010.279,A -85,B 0,C 180,E1 31324.774,E2 31324.774} C_VEL
LIN {X 0,Y 175.876,Z 1032.156,A -85,B 0,C 180,E1 31331.18,E2 31331.18} C_VEL
LIN {X 0,Y 144.392,Z 1044.615,A -85,B 0,C 180,E1 31335.011,E2 31335.011} C_VEL
LIN {X 0,Y 91.581,Z 1061.027,A -85,B 0,C 180,E1 31361.828,E2 31361.828} C_VEL
LIN {X 0,Y 74.574,Z 1064.676,A -85,B 0,C 180,E1 31404.162,E2 31404.162} C_VEL
LIN {X 0,Y 81.25,Z 1061.646,A -85,B 0,C 180,E1 31437.81,E2 31437.81} C_VEL
LIN {X 0,Y 126.926,Z 1045.261,A -85,B 0,C 180,E1 31473.639,E2 31473.639} C_VEL
LIN {X 0,Y 190.749,Z 1014.063,A -85,B 0,C 180,E1 31488.664,E2 31488.664} C_VEL
LIN {X 0,Y 252.884,Z 970.069,A -85,B 0,C 180,E1 31495.487,E2 31495.487} C_VEL
LIN {X 0,Y 267.585,Z 957.051,A -85,B 0,C 180,E1 31496.745,E2 31496.745} C_VEL
LIN {X 0,Y 268.184,Z 956.571,A -85,B 0,C 180,E1 31499.683,E2 31499.683} C_VEL
LIN {X 0,Y 205.753,Z 1005.247,A -85,B 0,C 180,E1 31505.765,E2 31505.765} C_VEL
LIN {X 0,Y 143.023,Z 1039.234,A -85,B 0,C 180,E1 31517.407,E2 31517.407} C_VEL
LIN {X 0,Y 92.848,Z 1058.801,A -85,B 0,C 180,E1 31542.7,E2 31542.7} C_VEL
LIN {X 0,Y 74.789,Z 1065.87,A -85,B 0,C 180,E1 31584.184,E2 31584.184} C_VEL
LIN {X 0,Y 79.56,Z 1065.029,A -85,B 0,C 180,E1 31618.46,E2 31618.46} C_VEL
LIN {X 0,Y 124.457,Z 1052.337,A -85,B 0,C 180,E1 31656.043,E2 31656.043} C_VEL
LIN {X 0,Y 191.53,Z 1024.279,A -85,B 0,C 180,E1 31671.765,E2 31671.765} C_VEL
LIN {X 0,Y 255.349,Z 984.445,A -85,B 0,C 180,E1 31678.902,E2 31678.902} C_VEL
LIN {X 0,Y 190.556,Z 1024.403,A -85,B 0,C 180,E1 31685.874,E2 31685.874} C_VEL
LIN {X 0,Y 144.392,Z 1044.615,A -85,B 0,C 180,E1 31695.011,E2 31695.011} C_VEL
LIN {X 0,Y 113.121,Z 1054.152,A -85,B 0,C 180,E1 31701.258,E2 31701.258} C_VEL
LIN {X 0,Y 71.562,Z 1063.993,A -85,B 0,C 180,E1 31738.008,E2 31738.008} C_VEL
LIN {X 0,Y 67.478,Z 1064.355,A -85,B 0,C 180,E1 31776.449,E2 31776.449} C_VEL
LIN {X 0,Y 94.72,Z 1055.42,A -85,B 0,C 180,E1 31823.171,E2 31823.171} C_VEL
LIN {X 0,Y 156.754,Z 1031.286,A -85,B 0,C 180,E1 31845.791,E2 31845.791} C_VEL
LIN {X 0,Y 222.677,Z 993.04,A -85,B 0,C 180,E1 31854.831,E2 31854.831} C_VEL
LIN {X 0,Y 262.686,Z 961.551,A -85,B 0,C 180,E1 31858.38,E2 31858.38} C_VEL
LIN {X 0,Y 200.005,Z 1008.196,A -85,B 0,C 180,E1 31864.036,E2 31864.036} C_VEL
LIN {X 0,Y 134.052,Z 1041.809,A -85,B 0,C 180,E1 31875.95,E2 31875.95} C_VEL
LIN {X 0,Y 83.007,Z 1060.063,A -85,B 0,C 180,E1 31903.055,E2 31903.055} C_VEL
LIN {X 0,Y 66.781,Z 1065.787,A -85,B 0,C 180,E1 31943.484,E2 31943.484} C_VEL
LIN {X 0,Y 72.503,Z 1064.964,A -85,B 0,C 180,E1 31981.529,E2 31981.529} C_VEL
LIN {X 0,Y 121.33,Z 1052.311,A -85,B 0,C 180,E1 32019.62,E2 32019.62} C_VEL
LIN {X 0,Y 190.52,Z 1024.304,A -85,B 0,C 180,E1 32034.231,E2 32034.231} C_VEL
LIN {X 0,Y 232.072,Z 1000.445,A -85,B 0,C 180,E1 32038.843,E2 32038.843} C_VEL
LIN {X 0,Y 164.323,Z 1036.007,A -85,B 0,C 180,E1 32047.225,E2 32047.225} C_VEL
LIN {X 0,Y 113.121,Z 1054.152,A -85,B 0,C 180,E1 32061.258,E2 32061.258} C_VEL
LIN {X 0,Y 83.012,Z 1060.743,A -85,B 0,C 180,E1 32071.731,E2 32071.731} C_VEL
LIN {X 0,Y 58.529,Z 1064.843,A -85,B 0,C 180,E1 32122.553,E2 32122.553} C_VEL
LIN {X 0,Y 67.353,Z 1061.854,A -85,B 0,C 180,E1 32164.25,E2 32164.25} C_VEL
LIN {X 0,Y 120.558,Z 1045.552,A -85,B 0,C 180,E1 32200.621,E2 32200.621} C_VEL
LIN {X 0,Y 188.362,Z 1014.39,A -85,B 0,C 180,E1 32213.557,E2 32213.557} C_VEL
LIN {X 0,Y 238.174,Z 981.627,A -85,B 0,C 180,E1 32218.214,E2 32218.214} C_VEL
LIN {X 0,Y 172.735,Z 1023.095,A -85,B 0,C 180,E1 32224.948,E2 32224.948} C_VEL
LIN {X 0,Y 105.274,Z 1051.527,A -85,B 0,C 180,E1 32241.223,E2 32241.223} C_VEL
LIN {X 0,Y 65.674,Z 1063.245,A -85,B 0,C 180,E1 32274.746,E2 32274.746} C_VEL
LIN {X 0,Y 58.952,Z 1066.046,A -85,B 0,C 180,E1 32317.393,E2 32317.393} C_VEL
LIN {X 0,Y 86.591,Z 1060.691,A -85,B 0,C 180,E1 32368.692,E2 32368.692} C_VEL
LIN {X 0,Y 152.126,Z 1040.82,A -85,B 0,C 180,E1 32391.33,E2 32391.33} C_VEL
LIN {X 0,Y 207.894,Z 1014.88,A -85,B 0,C 180,E1 32398.868,E2 32398.868} C_VEL
LIN {X 0,Y 140,Z 1044.996,A -85,B 0,C 180,E1 32408.577,E2 32408.577} C_VEL
LIN {X 0,Y 83.012,Z 1060.743,A -85,B 0,C 180,E1 32431.731,E2 32431.731} C_VEL
LIN {X 0,Y 57.04,Z 1064.237,A -85,B 0,C 180,E1 32451.743,E2 32451.743} C_VEL
LIN {X 0,Y 51.576,Z 1064.541,A -85,B 0,C 180,E1 32498.449,E2 32498.449} C_VEL
LIN {X 0,Y 85.919,Z 1055.67,A -85,B 0,C 180,E1 32551.936,E2 32551.936} C_VEL
LIN {X 0,Y 151.567,Z 1032.484,A -85,B 0,C 180,E1 32571.424,E2 32571.424} C_VEL
LIN {X 0,Y 208.33,Z 1002.292,A -85,B 0,C 180,E1 32577.958,E2 32577.958} C_VEL
LIN {X 0,Y 144.88,Z 1035.615,A -85,B 0,C 180,E1 32586.117,E2 32586.117} C_VEL
LIN {X 0,Y 78.193,Z 1058.427,A -85,B 0,C 180,E1 32609.232,E2 32609.232} C_VEL
LIN {X 0,Y 50.803,Z 1065.621,A -85,B 0,C 180,E1 32661.421,E2 32661.421} C_VEL
LIN {X 0,Y 59.198,Z 1064.834,A -85,B 0,C 180,E1 32709.826,E2 32709.826} C_VEL
LIN {X 0,Y 116.593,Z 1052.26,A -85,B 0,C 180,E1 32747.287,E2 32747.287} C_VEL
LIN {X 0,Y 183.936,Z 1026.941,A -85,B 0,C 180,E1 32758.852,E2 32758.852} C_VEL
LIN {X 0,Y 112.347,Z 1053.053,A -85,B 0,C 180,E1 32771.606,E2 32771.606} C_VEL
LIN {X 0,Y 58.259,Z 1064.123,A -85,B 0,C 180,E1 32809.4,E2 32809.4} C_VEL
LIN {X 0,Y 57.04,Z 1064.237,A -85,B 0,C 180,E1 32811.743,E2 32811.743} C_VEL
LIN {X 0,Y 42.427,Z 1064.818,A -85,B 0,C 180,E1 32850.215,E2 32850.215} C_VEL
LIN {X 0,Y 64.639,Z 1059.968,A -85,B 0,C 180,E1 32905.188,E2 32905.188} C_VEL
LIN {X 0,Y 130.426,Z 1040.728,A -85,B 0,C 180,E1 32931.203,E2 32931.203} C_VEL
LIN {X 0,Y 181.658,Z 1017.747,A -85,B 0,C 180,E1 32938.424,E2 32938.424} C_VEL
LIN {X 0,Y 111.368,Z 1047.727,A -85,B 0,C 180,E1 32949.196,E2 32949.196} C_VEL
LIN {X 0,Y 53.174,Z 1063.038,A -85,B 0,C 180,E1 32984.53,E2 32984.53} C_VEL
LIN {X 0,Y 42.983,Z 1065.88,A -85,B 0,C 180,E1 33040.165,E2 33040.165} C_VEL
LIN {X 0,Y 80.804,Z 1060.301,A -85,B 0,C 180,E1 33099.779,E2 33099.779} C_VEL
LIN {X 0,Y 152.025,Z 1040.272,A -85,B 0,C 180,E1 33117.82,E2 33117.82} C_VEL
LIN {X 0,Y 159.26,Z 1037.518,A -85,B 0,C 180,E1 33118.84,E2 33118.84} C_VEL
LIN {X 0,Y 86.512,Z 1058.808,A -85,B 0,C 180,E1 33135.398,E2 33135.398} C_VEL
LIN {X 0,Y 45.413,Z 1064.865,A -85,B 0,C 180,E1 33179.937,E2 33179.937} C_VEL
LIN {X 0,Y 42.427,Z 1064.818,A -85,B 0,C 180,E1 33210.215,E2 33210.215} C_VEL
LIN {X 0,Y 46.805,Z 1062.539,A -85,B 0,C 180,E1 33257.013,E2 33257.013} C_VEL
LIN {X 0,Y 111.15,Z 1047.121,A -85,B 0,C 180,E1 33291.525,E2 33291.525} C_VEL
LIN {X 0,Y 154.215,Z 1031.029,A -85,B 0,C 180,E1 33298.395,E2 33298.395} C_VEL
LIN {X 0,Y 85.202,Z 1054.932,A -85,B 0,C 180,E1 33311.807,E2 33311.807} C_VEL
LIN {X 0,Y 39.219,Z 1064.469,A -85,B 0,C 180,E1 33354.557,E2 33354.557} C_VEL
LIN {X 0,Y 35.056,Z 1065.796,A -85,B 0,C 180,E1 33402.497,E2 33402.497} C_VEL
LIN {X 0,Y 78.325,Z 1060.255,A -85,B 0,C 180,E1 33465.483,E2 33465.483} C_VEL
LIN {X 0,Y 133.99,Z 1046.392,A -85,B 0,C 180,E1 33478.791,E2 33478.791} C_VEL
LIN {X 0,Y 70.93,Z 1061.254,A -85,B 0,C 180,E1 33495.823,E2 33495.823} C_VEL
LIN {X 0,Y 34.574,Z 1065.094,A -85,B 0,C 180,E1 33557.326,E2 33557.326} C_VEL
LIN {X 0,Y 46.805,Z 1062.539,A -85,B 0,C 180,E1 33617.013,E2 33617.013} C_VEL
LIN {X 0,Y 68.987,Z 1057.885,A -85,B 0,C 180,E1 33644.952,E2 33644.952} C_VEL
LIN {X 0,Y 125.744,Z 1042.165,A -85,B 0,C 180,E1 33658.018,E2 33658.018} C_VEL
LIN {X 0,Y 55.834,Z 1060.725,A -85,B 0,C 180,E1 33678.1,E2 33678.1} C_VEL
LIN {X 0,Y 27.093,Z 1065.371,A -85,B 0,C 180,E1 33733.756,E2 33733.756} C_VEL
LIN {X 0,Y 43.288,Z 1064.639,A -85,B 0,C 180,E1 33811.147,E2 33811.147} C_VEL
LIN {X 0,Y 107.545,Z 1053.766,A -85,B 0,C 180,E1 33839.021,E2 33839.021} C_VEL
LIN {X 0,Y 42.627,Z 1064.318,A -85,B 0,C 180,E1 33867.198,E2 33867.198} C_VEL
LIN {X 0,Y 27.969,Z 1064.814,A -85,B 0,C 180,E1 33945.722,E2 33945.722} C_VEL
LIN {X 0,Y 68.987,Z 1057.885,A -85,B 0,C 180,E1 34004.952,E2 34004.952} C_VEL
LIN {X 0,Y 86.786,Z 1053.74,A -85,B 0,C 180,E1 34016.483,E2 34016.483} C_VEL
LIN {X 0,Y 96.447,Z 1051.293,A -85,B 0,C 180,E1 34018.154,E2 34018.154} C_VEL
LIN {X 0,Y 39.981,Z 1062.726,A -85,B 0,C 180,E1 34038.536,E2 34038.536} C_VEL
LIN {X 0,Y 19.607,Z 1065.63,A -85,B 0,C 180,E1 34132.761,E2 34132.761} C_VEL
LIN {X 0,Y 68.436,Z 1061.388,A -85,B 0,C 180,E1 34195.682,E2 34195.682} C_VEL
LIN {X 0,Y 79.514,Z 1059.562,A -85,B 0,C 180,E1 34199.343,E2 34199.343} C_VEL
LIN {X 0,Y 27.138,Z 1065.089,A -85,B 0,C 180,E1 34233.039,E2 34233.039} C_VEL
LIN {X 0,Y 20.351,Z 1064.902,A -85,B 0,C 180,E1 34311.863,E2 34311.863} C_VEL
LIN {X 0,Y 77.553,Z 1055.888,A -85,B 0,C 180,E1 34374.506,E2 34374.506} C_VEL
LIN {X 0,Y 86.786,Z 1053.74,A -85,B 0,C 180,E1 34376.483,E2 34376.483} C_VEL
LIN {X 0,Y 49.903,Z 1061.015,A -85,B 0,C 180,E1 34381.899,E2 34381.899} C_VEL
LIN {X 0,Y 12.425,Z 1065.204,A -85,B 0,C 180,E1 34432.415,E2 34432.415} C_VEL
LIN {X 0,Y 38.178,Z 1064.508,A -85,B 0,C 180,E1 34553.259,E2 34553.259} C_VEL
LIN {X 0,Y 50.576,Z 1063.475,A -85,B 0,C 180,E1 34559.497,E2 34559.497} C_VEL
LIN {X 0,Y 13.235,Z 1064.988,A -85,B 0,C 180,E1 34684.933,E2 34684.933} C_VEL
LIN {X 0,Y 61.365,Z 1059.145,A -85,B 0,C 180,E1 34738.774,E2 34738.774} C_VEL
LIN {X 0,Y 49.903,Z 1061.015,A -85,B 0,C 180,E1 34741.899,E2 34741.899} C_VEL
LIN {X 0,Y 10.984,Z 1064.895,A -85,B 0,C 180,E1 34746.46,E2 34746.46} C_VEL
LIN {X 0,Y 16.569,Z 1065.37,A -85,B 0,C 180,E1 34918.341,E2 34918.341} C_VEL
LIN {X 0,Y 8.089,Z 1065.073,A -85,B 0,C 180,E1 35079.54,E2 35079.54} C_VEL
LIN {X 0,Y 22.751,Z 1064.094,A -85,B 0,C 180,E1 35098.44,E2 35098.44} C_VEL
LIN {X 0,Y 10.984,Z 1064.895,A -85,B 0,C 180,E1 35106.46,E2 35106.46} C_VEL
LIN {X 0,Y 9.197,Z 1066.891,A -85,B 0,C 180,E1 35109.545,E2 35109.545} C_VEL
LIN {X 0,Y 9.197,Z 1075.5,A -85,B 0,C 180,E1 35109.545,E2 35109.545} C_VEL
LIN {X 0,Y 9.197,Z 1075.5,A -85,B 0,C 180,E1 35109.545,E2 35109.545}

QRS_NEXT_CUT()
PTP {E1 35097.324,E2 35097.324}
PTP {X 0,Y 759.833,A -85,B 0,C 180,E1 35097.324,E2 35097.324,E3 0,E4 0,E5 0,E6 0}
QRS_SPEED_INIT()
LIN {X 0,Y 759.833,Z 1075.5,A -85,B 0,C 180,E1 35097.324,E2 35097.324,E3 0,E4 0,E5 0,E6 0} C_VEL
LIN {X 0,Y 759.833,Z 261.401,A -85,B 0,C 180,E1 35097.324,E2 35097.324} C_VEL
LIN {X 0,Y 759.833,Z 253.323,A -85,B 0,C 180,E1 35097.324,E2 35097.324} C_VEL
LIN {X 0,Y 759.835,Z 251.323,A -85,B 0,C 180,E1 35097.174,E2 35097.174} C_VEL
LIN {X 0,Y 759.902,Z 251.32,A -85,B 0,C 180,E1 35094.488,E2 35094.488} C_VEL
LIN {X 0,Y 759.851,Z 251.325,A -85,B 0,C 180,E1 35091.601,E2 35091.601} C_VEL
LIN {X 0,Y 759.833,Z 251.324,A -85,B 0,C 180,E1 35089.153,E2 35089.153} C_VEL
LIN {X 0,Y 759.856,Z 251.321,A -85,B 0,C 180,E1 35086.686,E2 35086.686} C_VEL
LIN {X 0,Y 759.882,Z 251.326,A -85,B 0,C 180,E1 35083.723,E2 35083.723} C_VEL
LIN {X 0,Y 759.835,Z 251.324,A -85,B 0,C 180,E1 35081.192,E2 35081.192} C_VEL
LIN {X 0,Y 759.838,Z 251.322,A -85,B 0,C 180,E1 35078.784,E2 35078.784} C_VEL
LIN {X 0,Y 759.913,Z 251.321,A -85,B 0,C 180,E1 35076.092,E2 35076.092} C_VEL
LIN {X 0,Y 759.846,Z 251.324,A -85,B 0,C 180,E1 35073.253,E2 35073.253} C_VEL
LIN {X 0,Y 759.832,Z 251.324,A -85,B 0,C 180,E1 35070.863,E2 35070.863} C_VEL
LIN {X 0,Y 759.852,Z 251.322,A -85,B 0,C 180,E1 35068.417,E2 35068.417} C_VEL
LIN {X 0,Y 759.885,Z 251.327,A -85,B 0,C 180,E1 35065.45,E2 35065.45} C_VEL
LIN {X 0,Y 759.833,Z 251.324,A -85,B 0,C 180,E1 35062.842,E2 35062.842} C_VEL
LIN {X 0,Y 759.84,Z 251.323,A -85,B 0,C 180,E1 35060.438,E2 35060.438} C_VEL
LIN {X 0,Y 759.915,Z 251.324,A -85,B 0,C 180,E1 35057.648,E2 35057.648} C_VEL
LIN {X 0,Y 759.844,Z 251.326,A -85,B 0,C 180,E1 35054.93,E2 35054.93} C_VEL
LIN {X 0,Y 759.831,Z 251.324,A -85,B 0,C 180,E1 35052.53,E2 35052.53} C_VEL
LIN {X 0,Y 759.858,Z 251.322,A -85,B 0,C 180,E1 35050.051,E2 35050.051} C_VEL
LIN {X 0,Y 759.86,Z 251.318,A -85,B 0,C 180,E1 35046.967,E2 35046.967} C_VEL
LIN {X 0,Y 759.918,Z 251.488,A -85,B 0,C 180,E1 35045.515,E2 35045.515} C_VEL
LIN {X 0,Y 759.916,Z 257.485,A -85,B 0,C 180,E1 35045.072,E2 35045.072} C_VEL
LIN {X 0,Y 759.919,Z 277.935,A -85,B 0,C 180,E1 35043.711,E2 35043.711} C_VEL
LIN {X 0,Y 759.912,Z 524.409,A -85,B 0,C 180,E1 35040.907,E2 35040.907} C_VEL
LIN {X 0,Y 759.913,Z 709.377,A -85,B 0,C 180,E1 35038.846,E2 35038.846} C_VEL
LIN {X 0,Y 759.916,Z 728.46,A -85,B 0,C 180,E1 35038.552,E2 35038.552} C_VEL
LIN {X 0,Y 759.911,Z 750.266,A -85,B 0,C 180,E1 35038.118,E2 35038.118} C_VEL
LIN {X 0,Y 759.913,Z 776.516,A -85,B 0,C 180,E1 35037.442,E2 35037.442} C_VEL
LIN {X 0,Y 759.912,Z 796.129,A -85,B 0,C 180,E1 35036.828,E2 35036.828} C_VEL
LIN {X 0,Y 759.917,Z 815.883,A -85,B 0,C 180,E1 35036.112,E2 35036.112} C_VEL
LIN {X 0,Y 759.914,Z 836.087,A -85,B 0,C 180,E1 35035.276,E2 35035.276} C_VEL
LIN {X 0,Y 759.91,Z 860.356,A -85,B 0,C 180,E1 35034.114,E2 35034.114} C_VEL
LIN {X 0,Y 759.913,Z 879.174,A -85,B 0,C 180,E1 35033.085,E2 35033.085} C_VEL
LIN {X 0,Y 759.907,Z 898.196,A -85,B 0,C 180,E1 35031.929,E2 35031.929} C_VEL
LIN {X 0,Y 759.914,Z 919.387,A -85,B 0,C 180,E1 35030.471,E2 35030.471} C_VEL
LIN {X 0,Y 759.916,Z 935.812,A -85,B 0,C 180,E1 35029.205,E2 35029.205} C_VEL
LIN {X 0,Y 759.899,Z 954.318,A -85,B 0,C 180,E1 35027.616,E2 35027.616} C_VEL
LIN {X 0,Y 759.906,Z 969.706,A -85,B 0,C 180,E1 35026.119,E2 35026.119} C_VEL
LIN {X 0,Y 759.898,Z 984.161,A -85,B 0,C 180,E1 35024.556,E2 35024.556} C_VEL
LIN {X 0,Y 759.891,Z 998.608,A -85,B 0,C 180,E1 35022.771,E2 35022.771} C_VEL
LIN {X 0,Y 759.91,Z 1009.568,A -85,B 0,C 180,E1 35021.229,E2 35021.229} C_VEL
LIN {X 0,Y 759.907,Z 1019.661,A -85,B 0,C 180,E1 35019.62,E2 35019.62} C_VEL
LIN {X 0,Y 759.897,Z 1030.208,A -85,B 0,C 180,E1 35017.637,E2 35017.637} C_VEL
LIN {X 0,Y 759.915,Z 1037.555,A -85,B 0,C 180,E1 35015.966,E2 35015.966} C_VEL
LIN {X 0,Y 759.908,Z 1043.357,A -85,B 0,C 180,E1 35014.377,E2 35014.377} C_VEL
LIN {X 0,Y 759.89,Z 1048.831,A -85,B 0,C 180,E1 35012.489,E2 35012.489} C_VEL
LIN {X 0,Y 759.903,Z 1052.522,A -85,B 0,C 180,E1 35010.603,E2 35010.603} C_VEL
LIN {X 0,Y 759.916,Z 1054.479,A -85,B 0,C 180,E1 35009.02,E2 35009.02} C_VEL
LIN {X 0,Y 759.892,Z 1055.386,A -85,B 0,C 180,E1 35007.36,E2 35007.36} C_VEL
LIN {X 0,Y 759.891,Z 1054.862,A -85,B 0,C 180,E1 35005.321,E2 35005.321} C_VEL
LIN {X 0,Y 759.904,Z 1053.04,A -85,B 0,C 180,E1 35003.654,E2 35003.654} C_VEL
LIN {X 0,Y 759.901,Z 1050.186,A -85,B 0,C 180,E1 35002.059,E2 35002.059} C_VEL
LIN {X 0,Y 759.909,Z 1045.787,A -85,B 0,C 180,E1 35000.304,E2 35000.304} C_VEL
LIN {X 0,Y 759.89,Z 1039.016,A -85,B 0,C 180,E1 34998.309,E2 34998.309} C_VEL
LIN {X 0,Y 759.917,Z 1032.132,A -85,B 0,C 180,E1 34996.687,E2 34996.687} C_VEL
LIN {X 0,Y 759.892,Z 1024.36,A -85,B 0,C 180,E1 34995.132,E2 34995.132} C_VEL
LIN {X 0,Y 759.905,Z 1013.833,A -85,B 0,C 180,E1 34993.318,E2 34993.318} C_VEL
LIN {X 0,Y 759.903,Z 1001.372,A -85,B 0,C 180,E1 34991.512,E2 34991.512} C_VEL
LIN {X 0,Y 759.891,Z 990.191,A -85,B 0,C 180,E1 34990.074,E2 34990.074} C_VEL
LIN {X 0,Y 759.906,Z 975.459,A -85,B 0,C 180,E1 34988.382,E2 34988.382} C_VEL
LIN {X 0,Y 759.905,Z 959.147,A -85,B 0,C 180,E1 34986.75,E2 34986.75} C_VEL
LIN {X 0,Y 759.901,Z 943.1,A -85,B 0,C 180,E1 34985.306,E2 34985.306} C_VEL
LIN {X 0,Y 759.917,Z 923.73,A -85,B 0,C 180,E1 34983.762,E2 34983.762} C_VEL
LIN {X 0,Y 759.913,Z 906.557,A -85,B 0,C 180,E1 34982.536,E2 34982.536} C_VEL
LIN {X 0,Y 759.906,Z 885.069,A -85,B 0,C 180,E1 34981.164,E2 34981.164} C_VEL
LIN {X 0,Y 759.916,Z 865.048,A -85,B 0,C 180,E1 34980.044,E2 34980.044} C_VEL
LIN {X 0,Y 759.913,Z 846.751,A -85,B 0,C 180,E1 34979.126,E2 34979.126} C_VEL
LIN {X 0,Y 759.916,Z 823.974,A -85,B 0,C 180,E1 34978.112,E2 34978.112} C_VEL
LIN {X 0,Y 759.917,Z 800.283,A -85,B 0,C 180,E1 34977.224,E2 34977.224} C_VEL
LIN {X 0,Y 759.918,Z 781.304,A -85,B 0,C 180,E1 34976.611,E2 34976.611} C_VEL
LIN {X 0,Y 759.919,Z 762.511,A -85,B 0,C 180,E1 34976.09,E2 34976.09} C_VEL
LIN {X 0,Y 759.911,Z 743.9,A -85,B 0,C 180,E1 34975.656,E2 34975.656} C_VEL
LIN {X 0,Y 759.913,Z 724.022,A -85,B 0,C 180,E1 34975.282,E2 34975.282} C_VEL
LIN {X 0,Y 759.914,Z 701.343,A -85,B 0,C 180,E1 34974.96,E2 34974.96} C_VEL
LIN {X 0,Y 759.917,Z 451.179,A -85,B 0,C 180,E1 34972.182,E2 34972.182} C_VEL
LIN {X 0,Y 759.919,Z 277.686,A -85,B 0,C 180,E1 34970.189,E2 34970.189} C_VEL
LIN {X 0,Y 759.918,Z 251.561,A -85,B 0,C 180,E1 34968.411,E2 34968.411} C_VEL
LIN {X 0,Y 759.843,Z 251.322,A -85,B 0,C 180,E1 34965.714,E2 34965.714} C_VEL
LIN {X 0,Y 759.833,Z 251.324,A -85,B 0,C 180,E1 34963.283,E2 34963.283} C_VEL
LIN {X 0,Y 759.876,Z 251.327,A -85,B 0,C 180,E1 34960.718,E2 34960.718} C_VEL
LIN {X 0,Y 759.857,Z 251.321,A -85,B 0,C 180,E1 34957.727,E2 34957.727} C_VEL
LIN {X 0,Y 759.833,Z 251.324,A -85,B 0,C 180,E1 34955.289,E2 34955.289} C_VEL
LIN {X 0,Y 759.843,Z 251.325,A -85,B 0,C 180,E1 34952.907,E2 34952.907} C_VEL
LIN {X 0,Y 759.917,Z 251.321,A -85,B 0,C 180,E1 34950.028,E2 34950.028} C_VEL
LIN {X 0,Y 759.839,Z 251.322,A -85,B 0,C 180,E1 34947.339,E2 34947.339} C_VEL
LIN {X 0,Y 759.833,Z 251.323,A -85,B 0,C 180,E1 34944.951,E2 34944.951} C_VEL
LIN {X 0,Y 759.888,Z 251.327,A -85,B 0,C 180,E1 34942.327,E2 34942.327} C_VEL
LIN {X 0,Y 759.852,Z 251.321,A -85,B 0,C 180,E1 34939.366,E2 34939.366} C_VEL
LIN {X 0,Y 759.833,Z 251.324,A -85,B 0,C 180,E1 34936.927,E2 34936.927} C_VEL
LIN {X 0,Y 759.859,Z 251.325,A -85,B 0,C 180,E1 34934.422,E2 34934.422} C_VEL
LIN {X 0,Y 759.869,Z 251.321,A -85,B 0,C 180,E1 34931.384,E2 34931.384} C_VEL
LIN {X 0,Y 759.836,Z 251.323,A -85,B 0,C 180,E1 34928.933,E2 34928.933} C_VEL
LIN {X 0,Y 759.842,Z 251.323,A -85,B 0,C 180,E1 34926.498,E2 34926.498} C_VEL
LIN {X 0,Y 759.917,Z 251.323,A -85,B 0,C 180,E1 34923.697,E2 34923.697} C_VEL
LIN {X 0,Y 759.845,Z 251.321,A -85,B 0,C 180,E1 34920.98,E2 34920.98} C_VEL
LIN {X 0,Y 759.834,Z 251.323,A -85,B 0,C 180,E1 34918.567,E2 34918.567} C_VEL
LIN {X 0,Y 759.875,Z 251.326,A -85,B 0,C 180,E1 34916.001,E2 34916.001} C_VEL
LIN {X 0,Y 759.865,Z 251.32,A -85,B 0,C 180,E1 34913.047,E2 34913.047} C_VEL
LIN {X 0,Y 759.834,Z 251.323,A -85,B 0,C 180,E1 34910.532,E2 34910.532} C_VEL
LIN {X 0,Y 759.851,Z 251.325,A -85,B 0,C 180,E1 34908.077,E2 34908.077} C_VEL
LIN {X 0,Y 759.897,Z 251.32,A -85,B 0,C 180,E1 34905.132,E2 34905.132} C_VEL
LIN {X 0,Y 759.836,Z 251.323,A -85,B 0,C 180,E1 34902.461,E2 34902.461} C_VEL
LIN {X 0,Y 759.842,Z 251.324,A -85,B 0,C 180,E1 34900.073,E2 34900.073} C_VEL
LIN {X 0,Y 759.917,Z 251.324,A -85,B 0,C 180,E1 34897.274,E2 34897.274} C_VEL
LIN {X 0,Y 759.844,Z 251.322,A -85,B 0,C 180,E1 34894.513,E2 34894.513} C_VEL
LIN {X 0,Y 759.835,Z 251.324,A -85,B 0,C 180,E1 34892.15,E2 34892.15} C_VEL
LIN {X 0,Y 759.865,Z 251.326,A -85,B 0,C 180,E1 34889.649,E2 34889.649} C_VEL
LIN {X 0,Y 759.868,Z 251.32,A -85,B 0,C 180,E1 34886.63,E2 34886.63} C_VEL
LIN {X 0,Y 759.836,Z 251.323,A -85,B 0,C 180,E1 34884.155,E2 34884.155} C_VEL
LIN {X 0,Y 759.847,Z 251.324,A -85,B 0,C 180,E1 34881.699,E2 34881.699} C_VEL
LIN {X 0,Y 759.912,Z 251.321,A -85,B 0,C 180,E1 34878.819,E2 34878.819} C_VEL
LIN {X 0,Y 759.838,Z 251.323,A -85,B 0,C 180,E1 34876.092,E2 34876.092} C_VEL
LIN {X 0,Y 759.838,Z 251.324,A -85,B 0,C 180,E1 34873.698,E2 34873.698} C_VEL
LIN {X 0,Y 759.918,Z 251.319,A -85,B 0,C 180,E1 34870.939,E2 34870.939} C_VEL
LIN {X 0,Y 759.885,Z 251.572,A -85,B 0,C 180,E1 34869.168,E2 34869.168} C_VEL
LIN {X 0,Y 759.919,Z 265.631,A -85,B 0,C 180,E1 34868.201,E2 34868.201} C_VEL
LIN {X 0,Y 759.911,Z 287.746,A -85,B 0,C 180,E1 34866.759,E2 34866.759} C_VEL
LIN {X 0,Y 759.913,Z 509.631,A -85,B 0,C 180,E1 34864.229,E2 34864.229} C_VEL
LIN {X 0,Y 759.913,Z 719.586,A -85,B 0,C 180,E1 34861.888,E2 34861.888} C_VEL
LIN {X 0,Y 759.917,Z 739.486,A -85,B 0,C 180,E1 34861.58,E2 34861.58} C_VEL
LIN {X 0,Y 759.912,Z 763.973,A -85,B 0,C 180,E1 34861.083,E2 34861.083} C_VEL
LIN {X 0,Y 759.914,Z 786.92,A -85,B 0,C 180,E1 34860.475,E2 34860.475} C_VEL
LIN {X 0,Y 759.914,Z 806.787,A -85,B 0,C 180,E1 34859.851,E2 34859.851} C_VEL
LIN {X 0,Y 759.915,Z 825.386,A -85,B 0,C 180,E1 34859.176,E2 34859.176} C_VEL
LIN {X 0,Y 759.915,Z 845.187,A -85,B 0,C 180,E1 34858.359,E2 34858.359} C_VEL
LIN {X 0,Y 759.91,Z 869.747,A -85,B 0,C 180,E1 34857.191,E2 34857.191} C_VEL
LIN {X 0,Y 759.914,Z 888.762,A -85,B 0,C 180,E1 34856.154,E2 34856.154} C_VEL
LIN {X 0,Y 759.906,Z 907.367,A -85,B 0,C 180,E1 34855.026,E2 34855.026} C_VEL
LIN {X 0,Y 759.913,Z 929.1,A -85,B 0,C 180,E1 34853.537,E2 34853.537} C_VEL
LIN {X 0,Y 759.913,Z 946.087,A -85,B 0,C 180,E1 34852.228,E2 34852.228} C_VEL
LIN {X 0,Y 759.898,Z 964.448,A -85,B 0,C 180,E1 34850.649,E2 34850.649} C_VEL
LIN {X 0,Y 759.903,Z 980.083,A -85,B 0,C 180,E1 34849.125,E2 34849.125} C_VEL
LIN {X 0,Y 759.902,Z 994.731,A -85,B 0,C 180,E1 34847.537,E2 34847.537} C_VEL
LIN {X 0,Y 759.891,Z 1008.685,A -85,B 0,C 180,E1 34845.806,E2 34845.806} C_VEL
LIN {X 0,Y 759.91,Z 1019.249,A -85,B 0,C 180,E1 34844.322,E2 34844.322} C_VEL
LIN {X 0,Y 759.914,Z 1029.022,A -85,B 0,C 180,E1 34842.771,E2 34842.771} C_VEL
LIN {X 0,Y 759.897,Z 1039.449,A -85,B 0,C 180,E1 34840.846,E2 34840.846} C_VEL
LIN {X 0,Y 759.917,Z 1047.262,A -85,B 0,C 180,E1 34839.085,E2 34839.085} C_VEL
LIN {X 0,Y 759.908,Z 1053.146,A -85,B 0,C 180,E1 34837.485,E2 34837.485} C_VEL
LIN {X 0,Y 759.892,Z 1058.272,A -85,B 0,C 180,E1 34835.739,E2 34835.739} C_VEL
LIN {X 0,Y 759.907,Z 1062.449,A -85,B 0,C 180,E1 34833.697,E2 34833.697} C_VEL
LIN {X 0,Y 759.911,Z 1064.504,A -85,B 0,C 180,E1 34832.036,E2 34832.036} C_VEL
LIN {X 0,Y 759.892,Z 1065.395,A -85,B 0,C 180,E1 34830.377,E2 34830.377} C_VEL
LIN {X 0,Y 759.894,Z 1064.84,A -85,B 0,C 180,E1 34828.341,E2 34828.341} C_VEL
LIN {X 0,Y 759.903,Z 1063.013,A -85,B 0,C 180,E1 34826.681,E2 34826.681} C_VEL
LIN {X 0,Y 759.901,Z 1060.165,A -85,B 0,C 180,E1 34825.094,E2 34825.094} C_VEL
LIN {X 0,Y 759.908,Z 1055.792,A -85,B 0,C 180,E1 34823.351,E2 34823.351} C_VEL
LIN {X 0,Y 759.89,Z 1049.092,A -85,B 0,C 180,E1 34821.373,E2 34821.373} C_VEL
LIN {X 0,Y 759.919,Z 1042.298,A -85,B 0,C 180,E1 34819.768,E2 34819.768} C_VEL
LIN {X 0,Y 759.893,Z 1034.649,A -85,B 0,C 180,E1 34818.232,E2 34818.232} C_VEL
LIN {X 0,Y 759.905,Z 1024.384,A -85,B 0,C 180,E1 34816.455,E2 34816.455} C_VEL
LIN {X 0,Y 759.91,Z 1012.169,A -85,B 0,C 180,E1 34814.664,E2 34814.664} C_VEL
LIN {X 0,Y 759.89,Z 1000.629,A -85,B 0,C 180,E1 34813.173,E2 34813.173} C_VEL
LIN {X 0,Y 759.915,Z 986.71,A -85,B 0,C 180,E1 34811.566,E2 34811.566} C_VEL
LIN {X 0,Y 759.899,Z 970.411,A -85,B 0,C 180,E1 34809.914,E2 34809.914} C_VEL
LIN {X 0,Y 759.911,Z 955.307,A -85,B 0,C 180,E1 34808.544,E2 34808.544} C_VEL
LIN {X 0,Y 759.912,Z 936.29,A -85,B 0,C 180,E1 34806.996,E2 34806.996} C_VEL
LIN {X 0,Y 759.909,Z 917.988,A -85,B 0,C 180,E1 34805.679,E2 34805.679} C_VEL
LIN {X 0,Y 759.911,Z 898.103,A -85,B 0,C 180,E1 34804.39,E2 34804.39} C_VEL
LIN {X 0,Y 759.919,Z 876.005,A -85,B 0,C 180,E1 34803.139,E2 34803.139} C_VEL
LIN {X 0,Y 759.912,Z 857.306,A -85,B 0,C 180,E1 34802.197,E2 34802.197} C_VEL
LIN {X 0,Y 759.915,Z 836.246,A -85,B 0,C 180,E1 34801.255,E2 34801.255} C_VEL
LIN {X 0,Y 759.917,Z 811.548,A -85,B 0,C 180,E1 34800.312,E2 34800.312} C_VEL
LIN {X 0,Y 759.918,Z 791.896,A -85,B 0,C 180,E1 34799.673,E2 34799.673} C_VEL
LIN {X 0,Y 759.917,Z 773.019,A -85,B 0,C 180,E1 34799.148,E2 34799.148} C_VEL
LIN {X 0,Y 759.912,Z 754.182,A -85,B 0,C 180,E1 34798.708,E2 34798.708} C_VEL
LIN {X 0,Y 759.914,Z 734.31,A -85,B 0,C 180,E1 34798.332,E2 34798.332} C_VEL
LIN {X 0,Y 759.916,Z 712.596,A -85,B 0,C 180,E1 34798.021,E2 34798.021} C_VEL
LIN {X 0,Y 759.913,Z 458.882,A -85,B 0,C 180,E1 34795.201,E2 34795.201} C_VEL
LIN {X 0,Y 759.911,Z 287.544,A -85,B 0,C 180,E1 34793.232,E2 34793.232} C_VEL
LIN {X 0,Y 759.901,Z 252.603,A -85,B 0,C 180,E1 34790.926,E2 34790.926} C_VEL
LIN {X 0,Y 759.882,Z 251.494,A -85,B 0,C 180,E1 34790.809,E2 34790.809} C_VEL
LIN {X 0,Y 759.837,Z 251.324,A -85,B 0,C 180,E1 34788.252,E2 34788.252} C_VEL
LIN {X 0,Y 759.844,Z 251.322,A -85,B 0,C 180,E1 34785.822,E2 34785.822} C_VEL
LIN {X 0,Y 759.916,Z 251.324,A -85,B 0,C 180,E1 34783.071,E2 34783.071} C_VEL
LIN {X 0,Y 759.848,Z 251.325,A -85,B 0,C 180,E1 34780.348,E2 34780.348} C_VEL
LIN {X 0,Y 759.835,Z 251.323,A -85,B 0,C 180,E1 34777.919,E2 34777.919} C_VEL
LIN {X 0,Y 759.871,Z 251.321,A -85,B 0,C 180,E1 34775.379,E2 34775.379} C_VEL
LIN {X 0,Y 759.861,Z 251.326,A -85,B 0,C 180,E1 34772.35,E2 34772.35} C_VEL
LIN {X 0,Y 759.835,Z 251.323,A -85,B 0,C 180,E1 34769.866,E2 34769.866} C_VEL
LIN {X 0,Y 759.852,Z 251.321,A -85,B 0,C 180,E1 34767.424,E2 34767.424} C_VEL
LIN {X 0,Y 759.899,Z 251.327,A -85,B 0,C 180,E1 34764.487,E2 34764.487} C_VEL
LIN {X 0,Y 759.837,Z 251.324,A -85,B 0,C 180,E1 34761.864,E2 34761.864} C_VEL
LIN {X 0,Y 759.839,Z 251.323,A -85,B 0,C 180,E1 34759.447,E2 34759.447} C_VEL
LIN {X 0,Y 759.917,Z 251.322,A -85,B 0,C 180,E1 34756.669,E2 34756.669} C_VEL
LIN {X 0,Y 759.843,Z 251.325,A -85,B 0,C 180,E1 34753.857,E2 34753.857} C_VEL
LIN {X 0,Y 759.835,Z 251.323,A -85,B 0,C 180,E1 34751.461,E2 34751.461} C_VEL
LIN {X 0,Y 759.872,Z 251.321,A -85,B 0,C 180,E1 34748.933,E2 34748.933} C_VEL
LIN {X 0,Y 759.866,Z 251.326,A -85,B 0,C 180,E1 34745.967,E2 34745.967} C_VEL
LIN {X 0,Y 759.834,Z 251.324,A -85,B 0,C 180,E1 34743.47,E2 34743.47} C_VEL
LIN {X 0,Y 759.845,Z 251.322,A -85,B 0,C 180,E1 34741.056,E2 34741.056} C_VEL
LIN {X 0,Y 759.919,Z 251.327,A -85,B 0,C 180,E1 34738.19,E2 34738.19} C_VEL
LIN {X 0,Y 759.835,Z 251.323,A -85,B 0,C 180,E1 34737.174,E2 34737.174} C_VEL
LIN {X 0,Y 758.851,Z 251.451,A -85,B 0,C 180,E1 34736.593,E2 34736.593} C_VEL
LIN {X 0,Y 752.439,Z 252.246,A -85,B 0,C 180,E1 34734.967,E2 34734.967} C_VEL
LIN {X 0,Y 751.954,Z 252.309,A -85,B 0,C 180,E1 34734.544,E2 34734.544} C_VEL
LIN {X 0,Y 751.912,Z 252.313,A -85,B 0,C 180,E1 34731.589,E2 34731.589} C_VEL
LIN {X 0,Y 751.895,Z 252.313,A -85,B 0,C 180,E1 34729.115,E2 34729.115} C_VEL
LIN {X 0,Y 751.935,Z 252.309,A -85,B 0,C 180,E1 34726.543,E2 34726.543} C_VEL
LIN {X 0,Y 751.92,Z 252.314,A -85,B 0,C 180,E1 34723.546,E2 34723.546} C_VEL
LIN {X 0,Y 751.894,Z 252.313,A -85,B 0,C 180,E1 34721.066,E2 34721.066} C_VEL
LIN {X 0,Y 751.916,Z 252.31,A -85,B 0,C 180,E1 34718.567,E2 34718.567} C_VEL
LIN {X 0,Y 751.939,Z 252.313,A -85,B 0,C 180,E1 34715.572,E2 34715.572} C_VEL
LIN {X 0,Y 751.894,Z 252.31,A -85,B 0,C 180,E1 34712.996,E2 34712.996} C_VEL
LIN {X 0,Y 751.904,Z 252.312,A -85,B 0,C 180,E1 34710.577,E2 34710.577} C_VEL
LIN {X 0,Y 751.976,Z 252.314,A -85,B 0,C 180,E1 34707.744,E2 34707.744} C_VEL
LIN {X 0,Y 751.899,Z 252.314,A -85,B 0,C 180,E1 34705.001,E2 34705.001} C_VEL
LIN {X 0,Y 751.897,Z 252.312,A -85,B 0,C 180,E1 34702.574,E2 34702.574} C_VEL
LIN {X 0,Y 751.976,Z 252.31,A -85,B 0,C 180,E1 34699.842,E2 34699.842} C_VEL
LIN {X 0,Y 751.907,Z 252.314,A -85,B 0,C 180,E1 34696.985,E2 34696.985} C_VEL
LIN {X 0,Y 751.893,Z 252.314,A -85,B 0,C 180,E1 34694.537,E2 34694.537} C_VEL
LIN {X 0,Y 751.933,Z 252.312,A -85,B 0,C 180,E1 34691.979,E2 34691.979} C_VEL
LIN {X 0,Y 751.918,Z 252.315,A -85,B 0,C 180,E1 34688.975,E2 34688.975} C_VEL
LIN {X 0,Y 751.892,Z 252.294,A -85,B 0,C 180,E1 34686.561,E2 34686.561} C_VEL
LIN {X 0,Y 751.979,Z 252.644,A -85,B 0,C 180,E1 34685.901,E2 34685.901} C_VEL
LIN {X 0,Y 753.026,Z 255.618,A -85,B 0,C 180,E1 34685.614,E2 34685.614} C_VEL
LIN {X 0,Y 753.059,Z 278.157,A -85,B 0,C 180,E1 34684.098,E2 34684.098} C_VEL
LIN {X 0,Y 753.494,Z 281.329,A -85,B 0,C 180,E1 34684.03,E2 34684.03} C_VEL
LIN {X 0,Y 753.263,Z 533.143,A -85,B 0,C 180,E1 34681.149,E2 34681.149} C_VEL
LIN {X 0,Y 753.105,Z 709.885,A -85,B 0,C 180,E1 34679.162,E2 34679.162} C_VEL
LIN {X 0,Y 753.065,Z 730.769,A -85,B 0,C 180,E1 34678.833,E2 34678.833} C_VEL
LIN {X 0,Y 752.972,Z 757.495,A -85,B 0,C 180,E1 34678.266,E2 34678.266} C_VEL
LIN {X 0,Y 752.904,Z 778.464,A -85,B 0,C 180,E1 34677.698,E2 34677.698} C_VEL
LIN {X 0,Y 752.832,Z 797.207,A -85,B 0,C 180,E1 34677.101,E2 34677.101} C_VEL
LIN {X 0,Y 752.761,Z 816.836,A -85,B 0,C 180,E1 34676.379,E2 34676.379} C_VEL
LIN {X 0,Y 752.665,Z 840.128,A -85,B 0,C 180,E1 34675.396,E2 34675.396} C_VEL
LIN {X 0,Y 752.538,Z 862.49,A -85,B 0,C 180,E1 34674.288,E2 34674.288} C_VEL
LIN {X 0,Y 752.461,Z 881.221,A -85,B 0,C 180,E1 34673.245,E2 34673.245} C_VEL
LIN {X 0,Y 752.35,Z 902.923,A -85,B 0,C 180,E1 34671.888,E2 34671.888} C_VEL
LIN {X 0,Y 752.275,Z 921.809,A -85,B 0,C 180,E1 34670.542,E2 34670.542} C_VEL
LIN {X 0,Y 752.195,Z 940.47,A -85,B 0,C 180,E1 34669.067,E2 34669.067} C_VEL
LIN {X 0,Y 752.121,Z 958.034,A -85,B 0,C 180,E1 34667.485,E2 34667.485} C_VEL
LIN {X 0,Y 752.058,Z 973.106,A -85,B 0,C 180,E1 34665.975,E2 34665.975} C_VEL
LIN {X 0,Y 752.01,Z 989.038,A -85,B 0,C 180,E1 34664.161,E2 34664.161} C_VEL
LIN {X 0,Y 751.966,Z 1000.579,A -85,B 0,C 180,E1 34662.674,E2 34662.674} C_VEL
LIN {X 0,Y 751.96,Z 1011.527,A -85,B 0,C 180,E1 34661.088,E2 34661.088} C_VEL
LIN {X 0,Y 751.938,Z 1023.31,A -85,B 0,C 180,E1 34659.105,E2 34659.105} C_VEL
LIN {X 0,Y 751.917,Z 1031.42,A -85,B 0,C 180,E1 34657.488,E2 34657.488} C_VEL
LIN {X 0,Y 751.913,Z 1038.291,A -85,B 0,C 180,E1 34655.877,E2 34655.877} C_VEL
LIN {X 0,Y 751.916,Z 1044.988,A -85,B 0,C 180,E1 34653.965,E2 34653.965} C_VEL
LIN {X 0,Y 751.913,Z 1050.024,A -85,B 0,C 180,E1 34651.981,E2 34651.981} C_VEL
LIN {X 0,Y 751.9,Z 1052.907,A -85,B 0,C 180,E1 34650.381,E2 34650.381} C_VEL
LIN {X 0,Y 751.896,Z 1054.776,A -85,B 0,C 180,E1 34648.705,E2 34648.705} C_VEL
LIN {X 0,Y 751.895,Z 1055.416,A -85,B 0,C 180,E1 34646.646,E2 34646.646} C_VEL
LIN {X 0,Y 751.911,Z 1054.564,A -85,B 0,C 180,E1 34644.965,E2 34644.965} C_VEL
LIN {X 0,Y 751.904,Z 1052.652,A -85,B 0,C 180,E1 34643.356,E2 34643.356} C_VEL
LIN {X 0,Y 751.894,Z 1049.156,A -85,B 0,C 180,E1 34641.512,E2 34641.512} C_VEL
LIN {X 0,Y 751.914,Z 1043.779,A -85,B 0,C 180,E1 34639.581,E2 34639.581} C_VEL
LIN {X 0,Y 751.92,Z 1037.961,A -85,B 0,C 180,E1 34637.949,E2 34637.949} C_VEL
LIN {X 0,Y 751.913,Z 1030.897,A -85,B 0,C 180,E1 34636.308,E2 34636.308} C_VEL
LIN {X 0,Y 751.932,Z 1021.232,A -85,B 0,C 180,E1 34634.418,E2 34634.418} C_VEL
LIN {X 0,Y 751.964,Z 1010.528,A -85,B 0,C 180,E1 34632.671,E2 34632.671} C_VEL
LIN {X 0,Y 751.966,Z 999.935,A -85,B 0,C 180,E1 34631.149,E2 34631.149} C_VEL
LIN {X 0,Y 752.02,Z 986.633,A -85,B 0,C 180,E1 34629.451,E2 34629.451} C_VEL
LIN {X 0,Y 752.071,Z 971.032,A -85,B 0,C 180,E1 34627.721,E2 34627.721} C_VEL
LIN {X 0,Y 752.114,Z 956.152,A -85,B 0,C 180,E1 34626.246,E2 34626.246} C_VEL
LIN {X 0,Y 752.211,Z 937.148,A -85,B 0,C 180,E1 34624.574,E2 34624.574} C_VEL
LIN {X 0,Y 752.275,Z 920.611,A -85,B 0,C 180,E1 34623.278,E2 34623.278} C_VEL
LIN {X 0,Y 752.378,Z 900.34,A -85,B 0,C 180,E1 34621.85,E2 34621.85} C_VEL
LIN {X 0,Y 752.466,Z 879.997,A -85,B 0,C 180,E1 34620.594,E2 34620.594} C_VEL
LIN {X 0,Y 752.542,Z 861.102,A -85,B 0,C 180,E1 34619.548,E2 34619.548} C_VEL
LIN {X 0,Y 752.677,Z 836.378,A -85,B 0,C 180,E1 34618.35,E2 34618.35} C_VEL
LIN {X 0,Y 752.763,Z 815.588,A -85,B 0,C 180,E1 34617.482,E2 34617.482} C_VEL
LIN {X 0,Y 752.835,Z 795.685,A -85,B 0,C 180,E1 34616.757,E2 34616.757} C_VEL
LIN {X 0,Y 752.945,Z 771.628,A -85,B 0,C 180,E1 34616.008,E2 34616.008} C_VEL
LIN {X 0,Y 753.012,Z 747.214,A -85,B 0,C 180,E1 34615.408,E2 34615.408} C_VEL
LIN {X 0,Y 753.067,Z 727.013,A -85,B 0,C 180,E1 34615.012,E2 34615.012} C_VEL
LIN {X 0,Y 753.107,Z 707.688,A -85,B 0,C 180,E1 34614.719,E2 34614.719} C_VEL
LIN {X 0,Y 753.333,Z 449.417,A -85,B 0,C 180,E1 34611.814,E2 34611.814} C_VEL
LIN {X 0,Y 753.337,Z 279.346,A -85,B 0,C 180,E1 34609.847,E2 34609.847} C_VEL
LIN {X 0,Y 752.965,Z 277.08,A -85,B 0,C 180,E1 34609.756,E2 34609.756} C_VEL
LIN {X 0,Y 752.967,Z 255.304,A -85,B 0,C 180,E1 34608.271,E2 34608.271} C_VEL
LIN {X 0,Y 751.938,Z 252.398,A -85,B 0,C 180,E1 34607.961,E2 34607.961} C_VEL
LIN {X 0,Y 751.895,Z 252.313,A -85,B 0,C 180,E1 34605.462,E2 34605.462} C_VEL
LIN {X 0,Y 751.908,Z 252.314,A -85,B 0,C 180,E1 34603.015,E2 34603.015} C_VEL
LIN {X 0,Y 751.973,Z 252.31,A -85,B 0,C 180,E1 34600.132,E2 34600.132} C_VEL
LIN {X 0,Y 751.897,Z 252.311,A -85,B 0,C 180,E1 34597.426,E2 34597.426} C_VEL
LIN {X 0,Y 751.9,Z 252.314,A -85,B 0,C 180,E1 34594.999,E2 34594.999} C_VEL
LIN {X 0,Y 751.978,Z 252.313,A -85,B 0,C 180,E1 34592.222,E2 34592.222} C_VEL
LIN {X 0,Y 751.904,Z 252.311,A -85,B 0,C 180,E1 34589.423,E2 34589.423} C_VEL
LIN {X 0,Y 751.896,Z 252.313,A -85,B 0,C 180,E1 34587.004,E2 34587.004} C_VEL
LIN {X 0,Y 751.94,Z 252.313,A -85,B 0,C 180,E1 34584.428,E2 34584.428} C_VEL
LIN {X 0,Y 751.916,Z 252.31,A -85,B 0,C 180,E1 34581.433,E2 34581.433} C_VEL
LIN {X 0,Y 751.895,Z 252.311,A -85,B 0,C 180,E1 34578.934,E2 34578.934} C_VEL
LIN {X 0,Y 751.93,Z 252.315,A -85,B 0,C 180,E1 34576.374,E2 34576.374} C_VEL
LIN {X 0,Y 751.925,Z 252.308,A -85,B 0,C 180,E1 34573.378,E2 34573.378} C_VEL
LIN {X 0,Y 751.895,Z 252.312,A -85,B 0,C 180,E1 34570.885,E2 34570.885} C_VEL
LIN {X 0,Y 751.913,Z 252.314,A -85,B 0,C 180,E1 34568.411,E2 34568.411} C_VEL
LIN {X 0,Y 751.96,Z 252.309,A -85,B 0,C 180,E1 34565.494,E2 34565.494} C_VEL
LIN {X 0,Y 751.897,Z 252.312,A -85,B 0,C 180,E1 34562.82,E2 34562.82} C_VEL
LIN {X 0,Y 751.904,Z 252.311,A -85,B 0,C 180,E1 34560.381,E2 34560.381} C_VEL
LIN {X 0,Y 751.978,Z 252.312,A -85,B 0,C 180,E1 34557.561,E2 34557.561} C_VEL
LIN {X 0,Y 751.903,Z 252.311,A -85,B 0,C 180,E1 34554.812,E2 34554.812} C_VEL
LIN {X 0,Y 751.898,Z 252.31,A -85,B 0,C 180,E1 34552.358,E2 34552.358} C_VEL
LIN {X 0,Y 751.97,Z 252.317,A -85,B 0,C 180,E1 34549.659,E2 34549.659} C_VEL
LIN {X 0,Y 751.908,Z 252.308,A -85,B 0,C 180,E1 34546.758,E2 34546.758} C_VEL
LIN {X 0,Y 751.896,Z 252.312,A -85,B 0,C 180,E1 34544.32,E2 34544.32} C_VEL
LIN {X 0,Y 751.946,Z 252.316,A -85,B 0,C 180,E1 34541.7,E2 34541.7} C_VEL
LIN {X 0,Y 751.916,Z 252.309,A -85,B 0,C 180,E1 34538.713,E2 34538.713} C_VEL
LIN {X 0,Y 751.896,Z 252.313,A -85,B 0,C 180,E1 34536.238,E2 34536.238} C_VEL
LIN {X 0,Y 751.926,Z 252.315,A -85,B 0,C 180,E1 34533.716,E2 34533.716} C_VEL
LIN {X 0,Y 751.93,Z 252.31,A -85,B 0,C 180,E1 34530.702,E2 34530.702} C_VEL
LIN {X 0,Y 751.895,Z 252.311,A -85,B 0,C 180,E1 34528.185,E2 34528.185} C_VEL
LIN {X 0,Y 751.909,Z 252.312,A -85,B 0,C 180,E1 34525.77,E2 34525.77} C_VEL
LIN {X 0,Y 751.976,Z 252.306,A -85,B 0,C 180,E1 34522.866,E2 34522.866} C_VEL
LIN {X 0,Y 751.904,Z 252.312,A -85,B 0,C 180,E1 34520.231,E2 34520.231} C_VEL
LIN {X 0,Y 751.9,Z 252.314,A -85,B 0,C 180,E1 34517.791,E2 34517.791} C_VEL
LIN {X 0,Y 751.977,Z 252.316,A -85,B 0,C 180,E1 34515.084,E2 34515.084} C_VEL
LIN {X 0,Y 751.909,Z 252.312,A -85,B 0,C 180,E1 34512.186,E2 34512.186} C_VEL
LIN {X 0,Y 751.898,Z 252.308,A -85,B 0,C 180,E1 34509.765,E2 34509.765} C_VEL
LIN {X 0,Y 751.981,Z 252.794,A -85,B 0,C 180,E1 34509.562,E2 34509.562} C_VEL
LIN {X 0,Y 753.073,Z 256.236,A -85,B 0,C 180,E1 34509.247,E2 34509.247} C_VEL
LIN {X 0,Y 753.092,Z 288.125,A -85,B 0,C 180,E1 34507.141,E2 34507.141} C_VEL
LIN {X 0,Y 753.488,Z 291.368,A -85,B 0,C 180,E1 34507.075,E2 34507.075} C_VEL
LIN {X 0,Y 753.261,Z 541.457,A -85,B 0,C 180,E1 34504.214,E2 34504.214} C_VEL
LIN {X 0,Y 753.105,Z 719.76,A -85,B 0,C 180,E1 34502.209,E2 34502.209} C_VEL
LIN {X 0,Y 753.066,Z 740.459,A -85,B 0,C 180,E1 34501.884,E2 34501.884} C_VEL
LIN {X 0,Y 752.973,Z 766.622,A -85,B 0,C 180,E1 34501.334,E2 34501.334} C_VEL
LIN {X 0,Y 752.905,Z 788.965,A -85,B 0,C 180,E1 34500.728,E2 34500.728} C_VEL
LIN {X 0,Y 752.834,Z 807.509,A -85,B 0,C 180,E1 34500.135,E2 34500.135} C_VEL
LIN {X 0,Y 752.758,Z 827.224,A -85,B 0,C 180,E1 34499.409,E2 34499.409} C_VEL
LIN {X 0,Y 752.645,Z 851.041,A -85,B 0,C 180,E1 34498.399,E2 34498.399} C_VEL
LIN {X 0,Y 752.538,Z 872.621,A -85,B 0,C 180,E1 34497.326,E2 34497.326} C_VEL
LIN {X 0,Y 752.46,Z 891.674,A -85,B 0,C 180,E1 34496.263,E2 34496.263} C_VEL
LIN {X 0,Y 752.343,Z 913.759,A -85,B 0,C 180,E1 34494.875,E2 34494.875} C_VEL
LIN {X 0,Y 752.276,Z 932.246,A -85,B 0,C 180,E1 34493.554,E2 34493.554} C_VEL
LIN {X 0,Y 752.185,Z 951.121,A -85,B 0,C 180,E1 34492.057,E2 34492.057} C_VEL
LIN {X 0,Y 752.12,Z 967.856,A -85,B 0,C 180,E1 34490.547,E2 34490.547} C_VEL
LIN {X 0,Y 752.058,Z 982.936,A -85,B 0,C 180,E1 34489.037,E2 34489.037} C_VEL
LIN {X 0,Y 752.013,Z 998.701,A -85,B 0,C 180,E1 34487.248,E2 34487.248} C_VEL
LIN {X 0,Y 751.966,Z 1010.742,A -85,B 0,C 180,E1 34485.696,E2 34485.696} C_VEL
LIN {X 0,Y 751.96,Z 1021.855,A -85,B 0,C 180,E1 34484.084,E2 34484.084} C_VEL
LIN {X 0,Y 751.935,Z 1033.422,A -85,B 0,C 180,E1 34482.128,E2 34482.128} C_VEL
LIN {X 0,Y 751.917,Z 1041.587,A -85,B 0,C 180,E1 34480.497,E2 34480.497} C_VEL
LIN {X 0,Y 751.908,Z 1048.483,A -85,B 0,C 180,E1 34478.874,E2 34478.874} C_VEL
LIN {X 0,Y 751.914,Z 1055.171,A -85,B 0,C 180,E1 34476.95,E2 34476.95} C_VEL
LIN {X 0,Y 751.913,Z 1060.006,A -85,B 0,C 180,E1 34475.035,E2 34475.035} C_VEL
LIN {X 0,Y 751.901,Z 1062.9,A -85,B 0,C 180,E1 34473.431,E2 34473.431} C_VEL
LIN {X 0,Y 751.898,Z 1064.773,A -85,B 0,C 180,E1 34471.753,E2 34471.753} C_VEL
LIN {X 0,Y 751.895,Z 1065.417,A -85,B 0,C 180,E1 34469.695,E2 34469.695} C_VEL
LIN {X 0,Y 751.913,Z 1064.572,A -85,B 0,C 180,E1 34468.019,E2 34468.019} C_VEL
LIN {X 0,Y 751.903,Z 1062.675,A -85,B 0,C 180,E1 34466.417,E2 34466.417} C_VEL
LIN {X 0,Y 751.9,Z 1059.369,A -85,B 0,C 180,E1 34464.659,E2 34464.659} C_VEL
LIN {X 0,Y 751.913,Z 1053.912,A -85,B 0,C 180,E1 34462.666,E2 34462.666} C_VEL
LIN {X 0,Y 751.917,Z 1048.178,A -85,B 0,C 180,E1 34461.049,E2 34461.049} C_VEL
LIN {X 0,Y 751.914,Z 1041.231,A -85,B 0,C 180,E1 34459.426,E2 34459.426} C_VEL
LIN {X 0,Y 751.931,Z 1031.785,A -85,B 0,C 180,E1 34457.56,E2 34457.56} C_VEL
LIN {X 0,Y 751.962,Z 1020.814,A -85,B 0,C 180,E1 34455.759,E2 34455.759} C_VEL
LIN {X 0,Y 751.966,Z 1010.429,A -85,B 0,C 180,E1 34454.261,E2 34454.261} C_VEL
LIN {X 0,Y 752.018,Z 998.059,A -85,B 0,C 180,E1 34452.673,E2 34452.673} C_VEL
LIN {X 0,Y 752.066,Z 981.642,A -85,B 0,C 180,E1 34450.829,E2 34450.829} C_VEL
LIN {X 0,Y 752.115,Z 967.005,A -85,B 0,C 180,E1 34449.372,E2 34449.372} C_VEL
LIN {X 0,Y 752.208,Z 948.622,A -85,B 0,C 180,E1 34447.738,E2 34447.738} C_VEL
LIN {X 0,Y 752.274,Z 931.314,A -85,B 0,C 180,E1 34446.376,E2 34446.376} C_VEL
LIN {X 0,Y 752.373,Z 911.514,A -85,B 0,C 180,E1 34444.971,E2 34444.971} C_VEL
LIN {X 0,Y 752.464,Z 890.22,A -85,B 0,C 180,E1 34443.652,E2 34443.652} C_VEL
LIN {X 0,Y 752.542,Z 871.236,A -85,B 0,C 180,E1 34442.6,E2 34442.6} C_VEL
LIN {X 0,Y 752.676,Z 846.846,A -85,B 0,C 180,E1 34441.415,E2 34441.415} C_VEL
LIN {X 0,Y 752.761,Z 826.511,A -85,B 0,C 180,E1 34440.563,E2 34440.563} C_VEL
LIN {X 0,Y 752.834,Z 806.851,A -85,B 0,C 180,E1 34439.842,E2 34439.842} C_VEL
LIN {X 0,Y 752.913,Z 785.3,A -85,B 0,C 180,E1 34439.162,E2 34439.162} C_VEL
LIN {X 0,Y 753.011,Z 758.902,A -85,B 0,C 180,E1 34438.489,E2 34438.489} C_VEL
LIN {X 0,Y 753.068,Z 737.936,A -85,B 0,C 180,E1 34438.073,E2 34438.073} C_VEL
LIN {X 0,Y 753.107,Z 718.503,A -85,B 0,C 180,E1 34437.775,E2 34437.775} C_VEL
LIN {X 0,Y 753.333,Z 458.647,A -85,B 0,C 180,E1 34434.85,E2 34434.85} C_VEL
LIN {X 0,Y 753.353,Z 289.239,A -85,B 0,C 180,E1 34432.892,E2 34432.892} C_VEL
LIN {X 0,Y 752.967,Z 286.662,A -85,B 0,C 180,E1 34432.785,E2 34432.785} C_VEL
LIN {X 0,Y 753.037,Z 255.515,A -85,B 0,C 180,E1 34430.701,E2 34430.701} C_VEL
LIN {X 0,Y 751.928,Z 252.488,A -85,B 0,C 180,E1 34430.385,E2 34430.385} C_VEL
LIN {X 0,Y 751.899,Z 252.313,A -85,B 0,C 180,E1 34428.018,E2 34428.018} C_VEL
LIN {X 0,Y 751.963,Z 252.307,A -85,B 0,C 180,E1 34425.349,E2 34425.349} C_VEL
LIN {X 0,Y 751.914,Z 252.314,A -85,B 0,C 180,E1 34422.436,E2 34422.436} C_VEL
LIN {X 0,Y 751.897,Z 252.313,A -85,B 0,C 180,E1 34419.964,E2 34419.964} C_VEL
LIN {X 0,Y 751.931,Z 252.309,A -85,B 0,C 180,E1 34417.424,E2 34417.424} C_VEL
LIN {X 0,Y 751.925,Z 252.312,A -85,B 0,C 180,E1 34414.413,E2 34414.413} C_VEL
LIN {X 0,Y 751.897,Z 252.313,A -85,B 0,C 180,E1 34411.956,E2 34411.956} C_VEL
LIN {X 0,Y 751.912,Z 252.31,A -85,B 0,C 180,E1 34409.474,E2 34409.474} C_VEL
LIN {X 0,Y 751.961,Z 252.317,A -85,B 0,C 180,E1 34406.538,E2 34406.538} C_VEL
LIN {X 0,Y 751.9,Z 252.313,A -85,B 0,C 180,E1 34403.929,E2 34403.929} C_VEL
LIN {X 0,Y 751.899,Z 252.312,A -85,B 0,C 180,E1 34401.533,E2 34401.533} C_VEL
LIN {X 0,Y 751.979,Z 252.309,A -85,B 0,C 180,E1 34398.771,E2 34398.771} C_VEL
LIN {X 0,Y 751.905,Z 252.314,A -85,B 0,C 180,E1 34395.899,E2 34395.899} C_VEL
LIN {X 0,Y 751.897,Z 252.312,A -85,B 0,C 180,E1 34393.457,E2 34393.457} C_VEL
LIN {X 0,Y 751.957,Z 252.309,A -85,B 0,C 180,E1 34390.806,E2 34390.806} C_VEL
LIN {X 0,Y 751.914,Z 252.314,A -85,B 0,C 180,E1 34387.873,E2 34387.873} C_VEL
LIN {X 0,Y 751.895,Z 252.312,A -85,B 0,C 180,E1 34385.418,E2 34385.418} C_VEL
LIN {X 0,Y 751.925,Z 252.31,A -85,B 0,C 180,E1 34382.896,E2 34382.896} C_VEL
LIN {X 0,Y 751.924,Z 252.314,A -85,B 0,C 180,E1 34379.848,E2 34379.848} C_VEL
LIN {X 0,Y 751.895,Z 252.313,A -85,B 0,C 180,E1 34377.332,E2 34377.332} C_VEL
LIN {X 0,Y 751.913,Z 252.31,A -85,B 0,C 180,E1 34374.88,E2 34374.88} C_VEL
LIN {X 0,Y 751.954,Z 252.309,A -85,B 0,C 180,E1 34374.544,E2 34374.544} C_VEL
LIN {X 0,Y 751.036,Z 252.433,A -85,B 0,C 180,E1 34373.957,E2 34373.957} C_VEL
LIN {X 0,Y 744.495,Z 253.25,A -85,B 0,C 180,E1 34372.272,E2 34372.272} C_VEL
LIN {X 0,Y 744.009,Z 253.303,A -85,B 0,C 180,E1 34371.888,E2 34371.888} C_VEL
LIN {X 0,Y 743.957,Z 253.302,A -85,B 0,C 180,E1 34369.255,E2 34369.255} C_VEL
LIN {X 0,Y 743.969,Z 253.298,A -85,B 0,C 180,E1 34366.792,E2 34366.792} C_VEL
LIN {X 0,Y 744.033,Z 253.304,A -85,B 0,C 180,E1 34363.918,E2 34363.918} C_VEL
LIN {X 0,Y 743.958,Z 253.303,A -85,B 0,C 180,E1 34361.182,E2 34361.182} C_VEL
LIN {X 0,Y 743.96,Z 253.299,A -85,B 0,C 180,E1 34358.805,E2 34358.805} C_VEL
LIN {X 0,Y 744.039,Z 253.3,A -85,B 0,C 180,E1 34356.039,E2 34356.039} C_VEL
LIN {X 0,Y 743.964,Z 253.298,A -85,B 0,C 180,E1 34353.178,E2 34353.178} C_VEL
LIN {X 0,Y 743.955,Z 253.302,A -85,B 0,C 180,E1 34350.799,E2 34350.799} C_VEL
LIN {X 0,Y 743.989,Z 253.299,A -85,B 0,C 180,E1 34348.29,E2 34348.29} C_VEL
LIN {X 0,Y 743.982,Z 253.304,A -85,B 0,C 180,E1 34345.26,E2 34345.26} C_VEL
LIN {X 0,Y 743.955,Z 253.301,A -85,B 0,C 180,E1 34342.785,E2 34342.785} C_VEL
LIN {X 0,Y 743.97,Z 253.301,A -85,B 0,C 180,E1 34340.327,E2 34340.327} C_VEL
LIN {X 0,Y 744.015,Z 253.305,A -85,B 0,C 180,E1 34337.364,E2 34337.364} C_VEL
LIN {X 0,Y 743.957,Z 253.304,A -85,B 0,C 180,E1 34334.77,E2 34334.77} C_VEL
LIN {X 0,Y 743.956,Z 253.303,A -85,B 0,C 180,E1 34332.43,E2 34332.43} C_VEL
LIN {X 0,Y 744.022,Z 253.298,A -85,B 0,C 180,E1 34329.761,E2 34329.761} C_VEL
LIN {X 0,Y 743.966,Z 253.272,A -85,B 0,C 180,E1 34326.828,E2 34326.828} C_VEL
LIN {X 0,Y 744.016,Z 253.69,A -85,B 0,C 180,E1 34326.32,E2 34326.32} C_VEL
LIN {X 0,Y 746.144,Z 259.712,A -85,B 0,C 180,E1 34325.751,E2 34325.751} C_VEL
LIN {X 0,Y 746.123,Z 278.157,A -85,B 0,C 180,E1 34324.503,E2 34324.503} C_VEL
LIN {X 0,Y 747.098,Z 282.844,A -85,B 0,C 180,E1 34324.384,E2 34324.384} C_VEL
LIN {X 0,Y 746.634,Z 534.373,A -85,B 0,C 180,E1 34321.482,E2 34321.482} C_VEL
LIN {X 0,Y 746.321,Z 710.021,A -85,B 0,C 180,E1 34319.489,E2 34319.489} C_VEL
LIN {X 0,Y 746.236,Z 731.617,A -85,B 0,C 180,E1 34319.145,E2 34319.145} C_VEL
LIN {X 0,Y 746.05,Z 758.73,A -85,B 0,C 180,E1 34318.558,E2 34318.558} C_VEL
LIN {X 0,Y 745.914,Z 779.7,A -85,B 0,C 180,E1 34317.98,E2 34317.98} C_VEL
LIN {X 0,Y 745.766,Z 799.521,A -85,B 0,C 180,E1 34317.336,E2 34317.336} C_VEL
LIN {X 0,Y 745.596,Z 823.218,A -85,B 0,C 180,E1 34316.438,E2 34316.438} C_VEL
LIN {X 0,Y 745.342,Z 846.714,A -85,B 0,C 180,E1 34315.379,E2 34315.379} C_VEL
LIN {X 0,Y 745.168,Z 866.434,A -85,B 0,C 180,E1 34314.369,E2 34314.369} C_VEL
LIN {X 0,Y 744.932,Z 889.419,A -85,B 0,C 180,E1 34313.033,E2 34313.033} C_VEL
LIN {X 0,Y 744.763,Z 908.173,A -85,B 0,C 180,E1 34311.791,E2 34311.791} C_VEL
LIN {X 0,Y 744.62,Z 927.702,A -85,B 0,C 180,E1 34310.352,E2 34310.352} C_VEL
LIN {X 0,Y 744.417,Z 946.147,A -85,B 0,C 180,E1 34308.806,E2 34308.806} C_VEL
LIN {X 0,Y 744.311,Z 962.588,A -85,B 0,C 180,E1 34307.271,E2 34307.271} C_VEL
LIN {X 0,Y 744.187,Z 979.196,A -85,B 0,C 180,E1 34305.508,E2 34305.508} C_VEL
LIN {X 0,Y 744.095,Z 991.853,A -85,B 0,C 180,E1 34303.997,E2 34303.997} C_VEL
LIN {X 0,Y 744.052,Z 1005.387,A -85,B 0,C 180,E1 34302.18,E2 34302.18} C_VEL
LIN {X 0,Y 743.988,Z 1017.1,A -85,B 0,C 180,E1 34300.332,E2 34300.332} C_VEL
LIN {X 0,Y 743.946,Z 1025.917,A -85,B 0,C 180,E1 34298.736,E2 34298.736} C_VEL
LIN {X 0,Y 743.923,Z 1034.75,A -85,B 0,C 180,E1 34296.87,E2 34296.87} C_VEL
LIN {X 0,Y 743.916,Z 1042.053,A -85,B 0,C 180,E1 34294.935,E2 34294.935} C_VEL
LIN {X 0,Y 743.91,Z 1046.951,A -85,B 0,C 180,E1 34293.313,E2 34293.313} C_VEL
LIN {X 0,Y 743.892,Z 1050.886,A -85,B 0,C 180,E1 34291.617,E2 34291.617} C_VEL
LIN {X 0,Y 743.915,Z 1053.999,A -85,B 0,C 180,E1 34289.615,E2 34289.615} C_VEL
LIN {X 0,Y 743.901,Z 1055.271,A -85,B 0,C 180,E1 34287.766,E2 34287.766} C_VEL
LIN {X 0,Y 743.9,Z 1055.272,A -85,B 0,C 180,E1 34286.146,E2 34286.146} C_VEL
LIN {X 0,Y 743.913,Z 1053.928,A -85,B 0,C 180,E1 34284.214,E2 34284.214} C_VEL
LIN {X 0,Y 743.892,Z 1050.85,A -85,B 0,C 180,E1 34282.275,E2 34282.275} C_VEL
LIN {X 0,Y 743.914,Z 1046.958,A -85,B 0,C 180,E1 34280.6,E2 34280.6} C_VEL
LIN {X 0,Y 743.918,Z 1041.867,A -85,B 0,C 180,E1 34278.919,E2 34278.919} C_VEL
LIN {X 0,Y 743.935,Z 1033.984,A -85,B 0,C 180,E1 34276.871,E2 34276.871} C_VEL
LIN {X 0,Y 743.941,Z 1025.66,A -85,B 0,C 180,E1 34275.125,E2 34275.125} C_VEL
LIN {X 0,Y 743.986,Z 1016.798,A -85,B 0,C 180,E1 34273.526,E2 34273.526} C_VEL
LIN {X 0,Y 744.057,Z 1004.98,A -85,B 0,C 180,E1 34271.672,E2 34271.672} C_VEL
LIN {X 0,Y 744.094,Z 992.026,A -85,B 0,C 180,E1 34269.934,E2 34269.934} C_VEL
LIN {X 0,Y 744.187,Z 979.168,A -85,B 0,C 180,E1 34268.399,E2 34268.399} C_VEL
LIN {X 0,Y 744.308,Z 962.731,A -85,B 0,C 180,E1 34266.653,E2 34266.653} C_VEL
LIN {X 0,Y 744.419,Z 946.54,A -85,B 0,C 180,E1 34265.139,E2 34265.139} C_VEL
LIN {X 0,Y 744.617,Z 928.178,A -85,B 0,C 180,E1 34263.594,E2 34263.594} C_VEL
LIN {X 0,Y 744.759,Z 908.562,A -85,B 0,C 180,E1 34262.147,E2 34262.147} C_VEL
LIN {X 0,Y 744.922,Z 889.883,A -85,B 0,C 180,E1 34260.906,E2 34260.906} C_VEL
LIN {X 0,Y 745.166,Z 866.904,A -85,B 0,C 180,E1 34259.566,E2 34259.566} C_VEL
LIN {X 0,Y 745.339,Z 847.379,A -85,B 0,C 180,E1 34258.563,E2 34258.563} C_VEL
LIN {X 0,Y 745.551,Z 825.225,A -85,B 0,C 180,E1 34257.557,E2 34257.557} C_VEL
LIN {X 0,Y 745.765,Z 800.593,A -85,B 0,C 180,E1 34256.612,E2 34256.612} C_VEL
LIN {X 0,Y 745.913,Z 780.962,A -85,B 0,C 180,E1 34255.968,E2 34255.968} C_VEL
LIN {X 0,Y 746.045,Z 760.492,A -85,B 0,C 180,E1 34255.398,E2 34255.398} C_VEL
LIN {X 0,Y 746.216,Z 735.98,A -85,B 0,C 180,E1 34254.842,E2 34254.842} C_VEL
LIN {X 0,Y 746.318,Z 711.178,A -85,B 0,C 180,E1 34254.437,E2 34254.437} C_VEL
LIN {X 0,Y 746.449,Z 644.243,A -85,B 0,C 180,E1 34253.666,E2 34253.666} C_VEL
LIN {X 0,Y 746.783,Z 420.763,A -85,B 0,C 180,E1 34251.127,E2 34251.127} C_VEL
LIN {X 0,Y 746.926,Z 281.237,A -85,B 0,C 180,E1 34249.497,E2 34249.497} C_VEL
LIN {X 0,Y 746.03,Z 277.14,A -85,B 0,C 180,E1 34249.355,E2 34249.355} C_VEL
LIN {X 0,Y 746.115,Z 259.144,A -85,B 0,C 180,E1 34248.117,E2 34248.117} C_VEL
LIN {X 0,Y 743.977,Z 253.44,A -85,B 0,C 180,E1 34247.549,E2 34247.549} C_VEL
LIN {X 0,Y 743.959,Z 253.303,A -85,B 0,C 180,E1 34245.206,E2 34245.206} C_VEL
LIN {X 0,Y 744.033,Z 253.304,A -85,B 0,C 180,E1 34242.457,E2 34242.457} C_VEL
LIN {X 0,Y 743.964,Z 253.302,A -85,B 0,C 180,E1 34239.573,E2 34239.573} C_VEL
LIN {X 0,Y 743.958,Z 253.3,A -85,B 0,C 180,E1 34237.156,E2 34237.156} C_VEL
LIN {X 0,Y 744.021,Z 253.304,A -85,B 0,C 180,E1 34234.457,E2 34234.457} C_VEL
LIN {X 0,Y 743.97,Z 253.3,A -85,B 0,C 180,E1 34231.521,E2 34231.521} C_VEL
LIN {X 0,Y 743.956,Z 253.302,A -85,B 0,C 180,E1 34229.113,E2 34229.113} C_VEL
LIN {X 0,Y 743.986,Z 253.303,A -85,B 0,C 180,E1 34226.586,E2 34226.586} C_VEL
LIN {X 0,Y 743.983,Z 253.3,A -85,B 0,C 180,E1 34223.526,E2 34223.526} C_VEL
LIN {X 0,Y 743.956,Z 253.3,A -85,B 0,C 180,E1 34221.03,E2 34221.03} C_VEL
LIN {X 0,Y 743.974,Z 253.3,A -85,B 0,C 180,E1 34218.574,E2 34218.574} C_VEL
LIN {X 0,Y 744.01,Z 253.297,A -85,B 0,C 180,E1 34215.592,E2 34215.592} C_VEL
LIN {X 0,Y 743.957,Z 253.297,A -85,B 0,C 180,E1 34212.971,E2 34212.971} C_VEL
LIN {X 0,Y 743.967,Z 253.303,A -85,B 0,C 180,E1 34210.532,E2 34210.532} C_VEL
LIN {X 0,Y 744.039,Z 253.292,A -85,B 0,C 180,E1 34207.646,E2 34207.646} C_VEL
LIN {X 0,Y 743.961,Z 253.3,A -85,B 0,C 180,E1 34204.935,E2 34204.935} C_VEL
LIN {X 0,Y 743.959,Z 253.302,A -85,B 0,C 180,E1 34202.542,E2 34202.542} C_VEL
LIN {X 0,Y 744.037,Z 253.298,A -85,B 0,C 180,E1 34199.769,E2 34199.769} C_VEL
LIN {X 0,Y 743.969,Z 253.301,A -85,B 0,C 180,E1 34196.918,E2 34196.918} C_VEL
LIN {X 0,Y 743.958,Z 253.301,A -85,B 0,C 180,E1 34194.447,E2 34194.447} C_VEL
LIN {X 0,Y 744.015,Z 253.299,A -85,B 0,C 180,E1 34191.81,E2 34191.81} C_VEL
LIN {X 0,Y 743.973,Z 253.299,A -85,B 0,C 180,E1 34188.841,E2 34188.841} C_VEL
LIN {X 0,Y 743.958,Z 253.296,A -85,B 0,C 180,E1 34186.34,E2 34186.34} C_VEL
LIN {X 0,Y 744.014,Z 253.303,A -85,B 0,C 180,E1 34183.687,E2 34183.687} C_VEL
LIN {X 0,Y 743.98,Z 253.296,A -85,B 0,C 180,E1 34180.775,E2 34180.775} C_VEL
LIN {X 0,Y 743.957,Z 253.3,A -85,B 0,C 180,E1 34178.309,E2 34178.309} C_VEL
LIN {X 0,Y 743.982,Z 253.304,A -85,B 0,C 180,E1 34175.801,E2 34175.801} C_VEL
LIN {X 0,Y 743.989,Z 253.299,A -85,B 0,C 180,E1 34172.723,E2 34172.723} C_VEL
LIN {X 0,Y 743.958,Z 253.302,A -85,B 0,C 180,E1 34170.179,E2 34170.179} C_VEL
LIN {X 0,Y 743.982,Z 253.301,A -85,B 0,C 180,E1 34167.663,E2 34167.663} C_VEL
LIN {X 0,Y 743.991,Z 253.3,A -85,B 0,C 180,E1 34164.602,E2 34164.602} C_VEL
LIN {X 0,Y 743.959,Z 253.296,A -85,B 0,C 180,E1 34162.086,E2 34162.086} C_VEL
LIN {X 0,Y 743.974,Z 253.304,A -85,B 0,C 180,E1 34159.624,E2 34159.624} C_VEL
LIN {X 0,Y 744.016,Z 253.3,A -85,B 0,C 180,E1 34156.64,E2 34156.64} C_VEL
LIN {X 0,Y 743.959,Z 253.298,A -85,B 0,C 180,E1 34154.015,E2 34154.015} C_VEL
LIN {X 0,Y 743.971,Z 253.304,A -85,B 0,C 180,E1 34151.53,E2 34151.53} C_VEL
LIN {X 0,Y 743.998,Z 253.54,A -85,B 0,C 180,E1 34150.034,E2 34150.034} C_VEL
LIN {X 0,Y 746.245,Z 259.85,A -85,B 0,C 180,E1 34149.428,E2 34149.428} C_VEL
LIN {X 0,Y 746.18,Z 288.138,A -85,B 0,C 180,E1 34147.543,E2 34147.543} C_VEL
LIN {X 0,Y 747.092,Z 292.669,A -85,B 0,C 180,E1 34147.431,E2 34147.431} C_VEL
LIN {X 0,Y 746.636,Z 542.205,A -85,B 0,C 180,E1 34144.551,E2 34144.551} C_VEL
LIN {X 0,Y 746.321,Z 719.974,A -85,B 0,C 180,E1 34142.534,E2 34142.534} C_VEL
LIN {X 0,Y 746.237,Z 741.432,A -85,B 0,C 180,E1 34142.193,E2 34142.193} C_VEL
LIN {X 0,Y 746.05,Z 768.715,A -85,B 0,C 180,E1 34141.603,E2 34141.603} C_VEL
LIN {X 0,Y 745.914,Z 789.7,A -85,B 0,C 180,E1 34141.025,E2 34141.025} C_VEL
LIN {X 0,Y 745.766,Z 810.057,A -85,B 0,C 180,E1 34140.362,E2 34140.362} C_VEL
LIN {X 0,Y 745.575,Z 834.237,A -85,B 0,C 180,E1 34139.44,E2 34139.44} C_VEL
LIN {X 0,Y 745.343,Z 856.4,A -85,B 0,C 180,E1 34138.44,E2 34138.44} C_VEL
LIN {X 0,Y 745.17,Z 875.835,A -85,B 0,C 180,E1 34137.446,E2 34137.446} C_VEL
LIN {X 0,Y 744.961,Z 898.097,A -85,B 0,C 180,E1 34136.162,E2 34136.162} C_VEL
LIN {X 0,Y 744.761,Z 917.99,A -85,B 0,C 180,E1 34134.849,E2 34134.849} C_VEL
LIN {X 0,Y 744.625,Z 936.502,A -85,B 0,C 180,E1 34133.488,E2 34133.488} C_VEL
LIN {X 0,Y 744.421,Z 955.308,A -85,B 0,C 180,E1 34131.926,E2 34131.926} C_VEL
LIN {X 0,Y 744.331,Z 970.413,A -85,B 0,C 180,E1 34130.525,E2 34130.525} C_VEL
LIN {X 0,Y 744.185,Z 987.971,A -85,B 0,C 180,E1 34128.693,E2 34128.693} C_VEL
LIN {X 0,Y 744.1,Z 1001.275,A -85,B 0,C 180,E1 34127.114,E2 34127.114} C_VEL
LIN {X 0,Y 744.051,Z 1013.914,A -85,B 0,C 180,E1 34125.431,E2 34125.431} C_VEL
LIN {X 0,Y 743.984,Z 1026.241,A -85,B 0,C 180,E1 34123.524,E2 34123.524} C_VEL
LIN {X 0,Y 743.944,Z 1035.235,A -85,B 0,C 180,E1 34121.912,E2 34121.912} C_VEL
LIN {X 0,Y 743.945,Z 1043.012,A -85,B 0,C 180,E1 34120.297,E2 34120.297} C_VEL
LIN {X 0,Y 743.917,Z 1051.105,A -85,B 0,C 180,E1 34118.269,E2 34118.269} C_VEL
LIN {X 0,Y 743.92,Z 1056.619,A -85,B 0,C 180,E1 34116.483,E2 34116.483} C_VEL
LIN {X 0,Y 743.9,Z 1060.484,A -85,B 0,C 180,E1 34114.858,E2 34114.858} C_VEL
LIN {X 0,Y 743.911,Z 1063.352,A -85,B 0,C 180,E1 34113.159,E2 34113.159} C_VEL
LIN {X 0,Y 743.917,Z 1065.194,A -85,B 0,C 180,E1 34111.078,E2 34111.078} C_VEL
LIN {X 0,Y 743.892,Z 1065.328,A -85,B 0,C 180,E1 34109.384,E2 34109.384} C_VEL
LIN {X 0,Y 743.901,Z 1064.37,A -85,B 0,C 180,E1 34107.766,E2 34107.766} C_VEL
LIN {X 0,Y 743.91,Z 1061.884,A -85,B 0,C 180,E1 34105.838,E2 34105.838} C_VEL
LIN {X 0,Y 743.917,Z 1057.446,A -85,B 0,C 180,E1 34103.827,E2 34103.827} C_VEL
LIN {X 0,Y 743.923,Z 1052.636,A -85,B 0,C 180,E1 34102.198,E2 34102.198} C_VEL
LIN {X 0,Y 743.911,Z 1046.349,A -85,B 0,C 180,E1 34100.484,E2 34100.484} C_VEL
LIN {X 0,Y 743.959,Z 1037.106,A -85,B 0,C 180,E1 34098.448,E2 34098.448} C_VEL
LIN {X 0,Y 743.989,Z 1028.098,A -85,B 0,C 180,E1 34096.793,E2 34096.793} C_VEL
LIN {X 0,Y 744.002,Z 1018.211,A -85,B 0,C 180,E1 34095.206,E2 34095.206} C_VEL
LIN {X 0,Y 744.089,Z 1005.06,A -85,B 0,C 180,E1 34093.359,E2 34093.359} C_VEL
LIN {X 0,Y 744.174,Z 991.191,A -85,B 0,C 180,E1 34091.675,E2 34091.675} C_VEL
LIN {X 0,Y 744.252,Z 976.944,A -85,B 0,C 180,E1 34090.126,E2 34090.126} C_VEL
LIN {X 0,Y 744.419,Z 959.029,A -85,B 0,C 180,E1 34088.406,E2 34088.406} C_VEL
LIN {X 0,Y 744.526,Z 942.536,A -85,B 0,C 180,E1 34086.995,E2 34086.995} C_VEL
LIN {X 0,Y 744.745,Z 921.615,A -85,B 0,C 180,E1 34085.405,E2 34085.405} C_VEL
LIN {X 0,Y 744.901,Z 903.401,A -85,B 0,C 180,E1 34084.178,E2 34084.178} C_VEL
LIN {X 0,Y 745.13,Z 882.201,A -85,B 0,C 180,E1 34082.898,E2 34082.898} C_VEL
LIN {X 0,Y 745.322,Z 859.962,A -85,B 0,C 180,E1 34081.734,E2 34081.734} C_VEL
LIN {X 0,Y 745.489,Z 840.391,A -85,B 0,C 180,E1 34080.828,E2 34080.828} C_VEL
LIN {X 0,Y 745.739,Z 816.493,A -85,B 0,C 180,E1 34079.863,E2 34079.863} C_VEL
LIN {X 0,Y 745.908,Z 792.639,A -85,B 0,C 180,E1 34079.064,E2 34079.064} C_VEL
LIN {X 0,Y 746.041,Z 772.38,A -85,B 0,C 180,E1 34078.492,E2 34078.492} C_VEL
LIN {X 0,Y 746.159,Z 751.804,A -85,B 0,C 180,E1 34078.011,E2 34078.011} C_VEL
LIN {X 0,Y 746.308,Z 726.295,A -85,B 0,C 180,E1 34077.549,E2 34077.549} C_VEL
LIN {X 0,Y 746.393,Z 686.885,A -85,B 0,C 180,E1 34077.076,E2 34077.076} C_VEL
LIN {X 0,Y 746.787,Z 450.726,A -85,B 0,C 180,E1 34074.404,E2 34074.404} C_VEL
LIN {X 0,Y 746.955,Z 291.165,A -85,B 0,C 180,E1 34072.543,E2 34072.543} C_VEL
LIN {X 0,Y 746.077,Z 287.402,A -85,B 0,C 180,E1 34072.426,E2 34072.426} C_VEL
LIN {X 0,Y 746.147,Z 259.233,A -85,B 0,C 180,E1 34070.524,E2 34070.524} C_VEL
LIN {X 0,Y 743.992,Z 253.488,A -85,B 0,C 180,E1 34069.953,E2 34069.953} C_VEL
LIN {X 0,Y 744.01,Z 253.3,A -85,B 0,C 180,E1 34067.469,E2 34067.469} C_VEL
LIN {X 0,Y 743.984,Z 253.305,A -85,B 0,C 180,E1 34064.552,E2 34064.552} C_VEL
LIN {X 0,Y 743.958,Z 253.3,A -85,B 0,C 180,E1 34062.015,E2 34062.015} C_VEL
LIN {X 0,Y 744.001,Z 253.299,A -85,B 0,C 180,E1 34059.398,E2 34059.398} C_VEL
LIN {X 0,Y 743.981,Z 253.304,A -85,B 0,C 180,E1 34056.386,E2 34056.386} C_VEL
LIN {X 0,Y 743.957,Z 253.297,A -85,B 0,C 180,E1 34053.902,E2 34053.902} C_VEL
LIN {X 0,Y 743.979,Z 253.3,A -85,B 0,C 180,E1 34051.415,E2 34051.415} C_VEL
LIN {X 0,Y 743.998,Z 253.302,A -85,B 0,C 180,E1 34048.409,E2 34048.409} C_VEL
LIN {X 0,Y 743.958,Z 253.302,A -85,B 0,C 180,E1 34045.815,E2 34045.815} C_VEL
LIN {X 0,Y 743.974,Z 253.299,A -85,B 0,C 180,E1 34043.358,E2 34043.358} C_VEL
LIN {X 0,Y 744.024,Z 253.304,A -85,B 0,C 180,E1 34040.452,E2 34040.452} C_VEL
LIN {X 0,Y 743.959,Z 253.302,A -85,B 0,C 180,E1 34037.764,E2 34037.764} C_VEL
LIN {X 0,Y 743.964,Z 253.3,A -85,B 0,C 180,E1 34035.353,E2 34035.353} C_VEL
LIN {X 0,Y 744.04,Z 253.303,A -85,B 0,C 180,E1 34032.496,E2 34032.496} C_VEL
LIN {X 0,Y 743.963,Z 253.302,A -85,B 0,C 180,E1 34029.75,E2 34029.75} C_VEL
LIN {X 0,Y 743.959,Z 253.301,A -85,B 0,C 180,E1 34027.309,E2 34027.309} C_VEL
LIN {X 0,Y 744.037,Z 253.299,A -85,B 0,C 180,E1 34024.548,E2 34024.548} C_VEL
LIN {X 0,Y 743.968,Z 253.303,A -85,B 0,C 180,E1 34021.694,E2 34021.694} C_VEL
LIN {X 0,Y 743.958,Z 253.3,A -85,B 0,C 180,E1 34019.23,E2 34019.23} C_VEL
LIN {X 0,Y 744.011,Z 253.299,A -85,B 0,C 180,E1 34016.61,E2 34016.61} C_VEL
LIN {X 0,Y 743.977,Z 253.304,A -85,B 0,C 180,E1 34013.673,E2 34013.673} C_VEL
LIN {X 0,Y 744.009,Z 253.303,A -85,B 0,C 180,E1 34011.888,E2 34011.888} C_VEL
LIN {X 0,Y 742.963,Z 253.426,A -85,B 0,C 180,E1 34011.294,E2 34011.294} C_VEL
LIN {X 0,Y 736.548,Z 254.232,A -85,B 0,C 180,E1 34009.633,E2 34009.633} C_VEL
LIN {X 0,Y 736.017,Z 254.291,A -85,B 0,C 180,E1 34009.201,E2 34009.201} C_VEL
LIN {X 0,Y 736.036,Z 254.286,A -85,B 0,C 180,E1 34006.727,E2 34006.727} C_VEL
LIN {X 0,Y 736.069,Z 254.291,A -85,B 0,C 180,E1 34003.75,E2 34003.75} C_VEL
LIN {X 0,Y 736.019,Z 254.292,A -85,B 0,C 180,E1 34001.136,E2 34001.136} C_VEL
LIN {X 0,Y 736.032,Z 254.287,A -85,B 0,C 180,E1 33998.649,E2 33998.649} C_VEL
LIN {X 0,Y 736.08,Z 254.289,A -85,B 0,C 180,E1 33995.695,E2 33995.695} C_VEL
LIN {X 0,Y 736.017,Z 254.285,A -85,B 0,C 180,E1 33993.016,E2 33993.016} C_VEL
LIN {X 0,Y 736.029,Z 254.29,A -85,B 0,C 180,E1 33990.543,E2 33990.543} C_VEL
LIN {X 0,Y 736.092,Z 254.284,A -85,B 0,C 180,E1 33987.642,E2 33987.642} C_VEL
LIN {X 0,Y 736.02,Z 254.292,A -85,B 0,C 180,E1 33984.925,E2 33984.925} C_VEL
LIN {X 0,Y 736.022,Z 254.289,A -85,B 0,C 180,E1 33982.501,E2 33982.501} C_VEL
LIN {X 0,Y 736.1,Z 254.291,A -85,B 0,C 180,E1 33979.715,E2 33979.715} C_VEL
LIN {X 0,Y 736.021,Z 254.292,A -85,B 0,C 180,E1 33976.846,E2 33976.846} C_VEL
LIN {X 0,Y 736.022,Z 254.292,A -85,B 0,C 180,E1 33974.391,E2 33974.391} C_VEL
LIN {X 0,Y 736.103,Z 254.292,A -85,B 0,C 180,E1 33971.543,E2 33971.543} C_VEL
LIN {X 0,Y 736.023,Z 254.292,A -85,B 0,C 180,E1 33968.759,E2 33968.759} C_VEL
LIN {X 0,Y 736.055,Z 254.484,A -85,B 0,C 180,E1 33966.79,E2 33966.79} C_VEL
LIN {X 0,Y 739.268,Z 263.06,A -85,B 0,C 180,E1 33965.944,E2 33965.944} C_VEL
LIN {X 0,Y 739.238,Z 278.257,A -85,B 0,C 180,E1 33964.912,E2 33964.912} C_VEL
LIN {X 0,Y 740.729,Z 284.747,A -85,B 0,C 180,E1 33964.739,E2 33964.739} C_VEL
LIN {X 0,Y 740.032,Z 535.628,A -85,B 0,C 180,E1 33961.82,E2 33961.82} C_VEL
LIN {X 0,Y 739.562,Z 710.158,A -85,B 0,C 180,E1 33959.822,E2 33959.822} C_VEL
LIN {X 0,Y 739.428,Z 732.875,A -85,B 0,C 180,E1 33959.456,E2 33959.456} C_VEL
LIN {X 0,Y 739.151,Z 759.338,A -85,B 0,C 180,E1 33958.871,E2 33958.871} C_VEL
LIN {X 0,Y 738.945,Z 780.224,A -85,B 0,C 180,E1 33958.29,E2 33958.29} C_VEL
LIN {X 0,Y 738.719,Z 800.598,A -85,B 0,C 180,E1 33957.619,E2 33957.619} C_VEL
LIN {X 0,Y 738.408,Z 825.447,A -85,B 0,C 180,E1 33956.655,E2 33956.655} C_VEL
LIN {X 0,Y 738.076,Z 847.478,A -85,B 0,C 180,E1 33955.647,E2 33955.647} C_VEL
LIN {X 0,Y 737.811,Z 867.929,A -85,B 0,C 180,E1 33954.584,E2 33954.584} C_VEL
LIN {X 0,Y 737.435,Z 891.617,A -85,B 0,C 180,E1 33953.175,E2 33953.175} C_VEL
LIN {X 0,Y 737.202,Z 909.288,A -85,B 0,C 180,E1 33951.984,E2 33951.984} C_VEL
LIN {X 0,Y 736.961,Z 929.18,A -85,B 0,C 180,E1 33950.49,E2 33950.49} C_VEL
LIN {X 0,Y 736.686,Z 946.552,A -85,B 0,C 180,E1 33949.011,E2 33949.011} C_VEL
LIN {X 0,Y 736.529,Z 962.954,A -85,B 0,C 180,E1 33947.459,E2 33947.459} C_VEL
LIN {X 0,Y 736.323,Z 979.505,A -85,B 0,C 180,E1 33945.678,E2 33945.678} C_VEL
LIN {X 0,Y 736.203,Z 992.286,A -85,B 0,C 180,E1 33944.131,E2 33944.131} C_VEL
LIN {X 0,Y 736.113,Z 1006.13,A -85,B 0,C 180,E1 33942.234,E2 33942.234} C_VEL
LIN {X 0,Y 736.022,Z 1017.051,A -85,B 0,C 180,E1 33940.488,E2 33940.488} C_VEL
LIN {X 0,Y 735.969,Z 1025.689,A -85,B 0,C 180,E1 33938.91,E2 33938.91} C_VEL
LIN {X 0,Y 735.96,Z 1033.846,A -85,B 0,C 180,E1 33937.18,E2 33937.18} C_VEL
LIN {X 0,Y 735.926,Z 1041.909,A -85,B 0,C 180,E1 33935.067,E2 33935.067} C_VEL
LIN {X 0,Y 735.917,Z 1046.833,A -85,B 0,C 180,E1 33933.427,E2 33933.427} C_VEL
LIN {X 0,Y 735.9,Z 1050.636,A -85,B 0,C 180,E1 33931.791,E2 33931.791} C_VEL
LIN {X 0,Y 735.916,Z 1053.792,A -85,B 0,C 180,E1 33929.844,E2 33929.844} C_VEL
LIN {X 0,Y 735.905,Z 1055.258,A -85,B 0,C 180,E1 33927.82,E2 33927.82} C_VEL
LIN {X 0,Y 735.898,Z 1055.285,A -85,B 0,C 180,E1 33926.183,E2 33926.183} C_VEL
LIN {X 0,Y 735.915,Z 1054.035,A -85,B 0,C 180,E1 33924.308,E2 33924.308} C_VEL
LIN {X 0,Y 735.892,Z 1050.942,A -85,B 0,C 180,E1 33922.269,E2 33922.269} C_VEL
LIN {X 0,Y 735.917,Z 1047.004,A -85,B 0,C 180,E1 33920.547,E2 33920.547} C_VEL
LIN {X 0,Y 735.92,Z 1042.272,A -85,B 0,C 180,E1 33918.955,E2 33918.955} C_VEL
LIN {X 0,Y 735.94,Z 1034.903,A -85,B 0,C 180,E1 33916.966,E2 33916.966} C_VEL
LIN {X 0,Y 735.966,Z 1026.311,A -85,B 0,C 180,E1 33915.121,E2 33915.121} C_VEL
LIN {X 0,Y 736.025,Z 1017.536,A -85,B 0,C 180,E1 33913.505,E2 33913.505} C_VEL
LIN {X 0,Y 736.079,Z 1007.424,A -85,B 0,C 180,E1 33911.876,E2 33911.876} C_VEL
LIN {X 0,Y 736.194,Z 993.262,A -85,B 0,C 180,E1 33909.902,E2 33909.902} C_VEL
LIN {X 0,Y 736.324,Z 980.297,A -85,B 0,C 180,E1 33908.324,E2 33908.324} C_VEL
LIN {X 0,Y 736.507,Z 964.463,A -85,B 0,C 180,E1 33906.599,E2 33906.599} C_VEL
LIN {X 0,Y 736.685,Z 947.071,A -85,B 0,C 180,E1 33904.946,E2 33904.946} C_VEL
LIN {X 0,Y 736.968,Z 928.873,A -85,B 0,C 180,E1 33903.395,E2 33903.395} C_VEL
LIN {X 0,Y 737.2,Z 909.255,A -85,B 0,C 180,E1 33901.924,E2 33901.924} C_VEL
LIN {X 0,Y 737.458,Z 890.629,A -85,B 0,C 180,E1 33900.671,E2 33900.671} C_VEL
LIN {X 0,Y 737.817,Z 867.006,A -85,B 0,C 180,E1 33899.276,E2 33899.276} C_VEL
LIN {X 0,Y 738.076,Z 847.098,A -85,B 0,C 180,E1 33898.244,E2 33898.244} C_VEL
LIN {X 0,Y 738.44,Z 824.32,A -85,B 0,C 180,E1 33897.206,E2 33897.206} C_VEL
LIN {X 0,Y 738.724,Z 799.98,A -85,B 0,C 180,E1 33896.27,E2 33896.27} C_VEL
LIN {X 0,Y 738.953,Z 779.657,A -85,B 0,C 180,E1 33895.603,E2 33895.603} C_VEL
LIN {X 0,Y 739.177,Z 756.554,A -85,B 0,C 180,E1 33894.966,E2 33894.966} C_VEL
LIN {X 0,Y 739.436,Z 730.415,A -85,B 0,C 180,E1 33894.411,E2 33894.411} C_VEL
LIN {X 0,Y 739.562,Z 709.506,A -85,B 0,C 180,E1 33894.08,E2 33894.08} C_VEL
LIN {X 0,Y 740.254,Z 453.575,A -85,B 0,C 180,E1 33891.147,E2 33891.147} C_VEL
LIN {X 0,Y 740.568,Z 283.278,A -85,B 0,C 180,E1 33889.144,E2 33889.144} C_VEL
LIN {X 0,Y 739.133,Z 277.34,A -85,B 0,C 180,E1 33888.954,E2 33888.954} C_VEL
LIN {X 0,Y 739.089,Z 262.381,A -85,B 0,C 180,E1 33887.907,E2 33887.907} C_VEL
LIN {X 0,Y 736.065,Z 254.546,A -85,B 0,C 180,E1 33887.136,E2 33887.136} C_VEL
LIN {X 0,Y 736.036,Z 254.288,A -85,B 0,C 180,E1 33885.822,E2 33885.822} C_VEL
LIN {X 0,Y 736.018,Z 254.29,A -85,B 0,C 180,E1 33883.319,E2 33883.319} C_VEL
LIN {X 0,Y 736.063,Z 254.293,A -85,B 0,C 180,E1 33880.696,E2 33880.696} C_VEL
LIN {X 0,Y 736.036,Z 254.286,A -85,B 0,C 180,E1 33877.685,E2 33877.685} C_VEL
LIN {X 0,Y 736.017,Z 254.292,A -85,B 0,C 180,E1 33875.266,E2 33875.266} C_VEL
LIN {X 0,Y 736.038,Z 254.292,A -85,B 0,C 180,E1 33872.766,E2 33872.766} C_VEL
LIN {X 0,Y 736.057,Z 254.288,A -85,B 0,C 180,E1 33869.725,E2 33869.725} C_VEL
LIN {X 0,Y 736.018,Z 254.29,A -85,B 0,C 180,E1 33867.149,E2 33867.149} C_VEL
LIN {X 0,Y 736.037,Z 254.287,A -85,B 0,C 180,E1 33864.649,E2 33864.649} C_VEL
LIN {X 0,Y 736.058,Z 254.286,A -85,B 0,C 180,E1 33861.601,E2 33861.601} C_VEL
LIN {X 0,Y 736.018,Z 254.286,A -85,B 0,C 180,E1 33859,E2 33859} C_VEL
LIN {X 0,Y 736.044,Z 254.293,A -85,B 0,C 180,E1 33856.449,E2 33856.449} C_VEL
LIN {X 0,Y 736.044,Z 254.283,A -85,B 0,C 180,E1 33853.352,E2 33853.352} C_VEL
LIN {X 0,Y 736.018,Z 254.291,A -85,B 0,C 180,E1 33850.827,E2 33850.827} C_VEL
LIN {X 0,Y 736.048,Z 254.292,A -85,B 0,C 180,E1 33848.279,E2 33848.279} C_VEL
LIN {X 0,Y 736.045,Z 254.287,A -85,B 0,C 180,E1 33845.222,E2 33845.222} C_VEL
LIN {X 0,Y 736.018,Z 254.291,A -85,B 0,C 180,E1 33842.725,E2 33842.725} C_VEL
LIN {X 0,Y 736.039,Z 254.287,A -85,B 0,C 180,E1 33840.234,E2 33840.234} C_VEL
LIN {X 0,Y 736.059,Z 254.289,A -85,B 0,C 180,E1 33837.197,E2 33837.197} C_VEL
LIN {X 0,Y 736.019,Z 254.288,A -85,B 0,C 180,E1 33834.621,E2 33834.621} C_VEL
LIN {X 0,Y 736.037,Z 254.284,A -85,B 0,C 180,E1 33832.114,E2 33832.114} C_VEL
LIN {X 0,Y 736.067,Z 254.287,A -85,B 0,C 180,E1 33829.116,E2 33829.116} C_VEL
LIN {X 0,Y 736.018,Z 254.283,A -85,B 0,C 180,E1 33826.487,E2 33826.487} C_VEL
LIN {X 0,Y 736.037,Z 254.29,A -85,B 0,C 180,E1 33823.992,E2 33823.992} C_VEL
LIN {X 0,Y 736.065,Z 254.283,A -85,B 0,C 180,E1 33820.972,E2 33820.972} C_VEL
LIN {X 0,Y 736.02,Z 254.287,A -85,B 0,C 180,E1 33818.398,E2 33818.398} C_VEL
LIN {X 0,Y 736.033,Z 254.293,A -85,B 0,C 180,E1 33815.909,E2 33815.909} C_VEL
LIN {X 0,Y 736.079,Z 254.287,A -85,B 0,C 180,E1 33812.931,E2 33812.931} C_VEL
LIN {X 0,Y 736.021,Z 254.291,A -85,B 0,C 180,E1 33810.274,E2 33810.274} C_VEL
LIN {X 0,Y 736.029,Z 254.289,A -85,B 0,C 180,E1 33807.815,E2 33807.815} C_VEL
LIN {X 0,Y 736.094,Z 254.289,A -85,B 0,C 180,E1 33804.929,E2 33804.929} C_VEL
LIN {X 0,Y 736.023,Z 254.283,A -85,B 0,C 180,E1 33802.216,E2 33802.216} C_VEL
LIN {X 0,Y 736.027,Z 254.293,A -85,B 0,C 180,E1 33799.771,E2 33799.771} C_VEL
LIN {X 0,Y 736.099,Z 254.29,A -85,B 0,C 180,E1 33796.953,E2 33796.953} C_VEL
LIN {X 0,Y 736.028,Z 254.286,A -85,B 0,C 180,E1 33794.169,E2 33794.169} C_VEL
LIN {X 0,Y 736.021,Z 254.292,A -85,B 0,C 180,E1 33791.733,E2 33791.733} C_VEL
LIN {X 0,Y 736.1,Z 254.491,A -85,B 0,C 180,E1 33790.488,E2 33790.488} C_VEL
LIN {X 0,Y 739.393,Z 263.101,A -85,B 0,C 180,E1 33789.639,E2 33789.639} C_VEL
LIN {X 0,Y 739.26,Z 287.971,A -85,B 0,C 180,E1 33787.96,E2 33787.96} C_VEL
LIN {X 0,Y 740.725,Z 294.467,A -85,B 0,C 180,E1 33787.788,E2 33787.788} C_VEL
LIN {X 0,Y 740.035,Z 543.581,A -85,B 0,C 180,E1 33784.888,E2 33784.888} C_VEL
LIN {X 0,Y 739.562,Z 720.082,A -85,B 0,C 180,E1 33782.868,E2 33782.868} C_VEL
LIN {X 0,Y 739.43,Z 742.404,A -85,B 0,C 180,E1 33782.509,E2 33782.509} C_VEL
LIN {X 0,Y 739.151,Z 769.149,A -85,B 0,C 180,E1 33781.921,E2 33781.921} C_VEL
LIN {X 0,Y 738.945,Z 790.438,A -85,B 0,C 180,E1 33781.328,E2 33781.328} C_VEL
LIN {X 0,Y 738.717,Z 811.333,A -85,B 0,C 180,E1 33780.638,E2 33780.638} C_VEL
LIN {X 0,Y 738.388,Z 836.243,A -85,B 0,C 180,E1 33779.666,E2 33779.666} C_VEL
LIN {X 0,Y 738.075,Z 857.294,A -85,B 0,C 180,E1 33778.702,E2 33778.702} C_VEL
LIN {X 0,Y 737.814,Z 877.443,A -85,B 0,C 180,E1 33777.656,E2 33777.656} C_VEL
LIN {X 0,Y 737.455,Z 900.756,A -85,B 0,C 180,E1 33776.276,E2 33776.276} C_VEL
LIN {X 0,Y 737.2,Z 919.199,A -85,B 0,C 180,E1 33775.035,E2 33775.035} C_VEL
LIN {X 0,Y 736.966,Z 938.96,A -85,B 0,C 180,E1 33773.553,E2 33773.553} C_VEL
LIN {X 0,Y 736.685,Z 956.907,A -85,B 0,C 180,E1 33772.024,E2 33772.024} C_VEL
LIN {X 0,Y 736.517,Z 973.81,A -85,B 0,C 180,E1 33770.42,E2 33770.42} C_VEL
LIN {X 0,Y 736.323,Z 989.775,A -85,B 0,C 180,E1 33768.692,E2 33768.692} C_VEL
LIN {X 0,Y 736.2,Z 1002.563,A -85,B 0,C 180,E1 33767.141,E2 33767.141} C_VEL
LIN {X 0,Y 736.101,Z 1016.649,A -85,B 0,C 180,E1 33765.198,E2 33765.198} C_VEL
LIN {X 0,Y 736.023,Z 1027.17,A -85,B 0,C 180,E1 33763.513,E2 33763.513} C_VEL
LIN {X 0,Y 735.969,Z 1035.879,A -85,B 0,C 180,E1 33761.918,E2 33761.918} C_VEL
LIN {X 0,Y 735.948,Z 1044.436,A -85,B 0,C 180,E1 33760.094,E2 33760.094} C_VEL
LIN {X 0,Y 735.929,Z 1051.871,A -85,B 0,C 180,E1 33758.123,E2 33758.123} C_VEL
LIN {X 0,Y 735.921,Z 1056.826,A -85,B 0,C 180,E1 33756.475,E2 33756.475} C_VEL
LIN {X 0,Y 735.899,Z 1060.643,A -85,B 0,C 180,E1 33754.832,E2 33754.832} C_VEL
LIN {X 0,Y 735.915,Z 1063.803,A -85,B 0,C 180,E1 33752.882,E2 33752.882} C_VEL
LIN {X 0,Y 735.904,Z 1065.261,A -85,B 0,C 180,E1 33750.856,E2 33750.856} C_VEL
LIN {X 0,Y 735.899,Z 1065.283,A -85,B 0,C 180,E1 33749.222,E2 33749.222} C_VEL
LIN {X 0,Y 735.914,Z 1064.035,A -85,B 0,C 180,E1 33747.352,E2 33747.352} C_VEL
LIN {X 0,Y 735.893,Z 1060.961,A -85,B 0,C 180,E1 33745.324,E2 33745.324} C_VEL
LIN {X 0,Y 735.918,Z 1057.033,A -85,B 0,C 180,E1 33743.603,E2 33743.603} C_VEL
LIN {X 0,Y 735.923,Z 1052.126,A -85,B 0,C 180,E1 33741.955,E2 33741.955} C_VEL
LIN {X 0,Y 735.94,Z 1044.789,A -85,B 0,C 180,E1 33739.985,E2 33739.985} C_VEL
LIN {X 0,Y 735.967,Z 1036.289,A -85,B 0,C 180,E1 33738.162,E2 33738.162} C_VEL
LIN {X 0,Y 736.025,Z 1027.635,A -85,B 0,C 180,E1 33736.567,E2 33736.567} C_VEL
LIN {X 0,Y 736.074,Z 1017.692,A -85,B 0,C 180,E1 33734.962,E2 33734.962} C_VEL
LIN {X 0,Y 736.193,Z 1003.471,A -85,B 0,C 180,E1 33732.974,E2 33732.974} C_VEL
